LIN {X 0,Y 445.736,Z 432.603,A -85,B 0,C 180,E1 -8644.071,E2 -8644.071} C_VEL
LIN {X 0,Y 445.822,Z 429.975,A -85,B 0,C 180,E1 -8644.977,E2 -8644.977} C_VEL
LIN {X 0,Y 445.879,Z 426.705,A -85,B 0,C 180,E1 -8645.883,E2 -8645.883} C_VEL
LIN {X 0,Y 446.166,Z 422.759,A -85,B 0,C 180,E1 -8646.774,E2 -8646.774} C_VEL
LIN {X 0,Y 446.258,Z 417.856,A -85,B 0,C 180,E1 -8647.696,E2 -8647.696} C_VEL
LIN {X 0,Y 446.578,Z 411.998,A -85,B 0,C 180,E1 -8648.601,E2 -8648.601} C_VEL
LIN {X 0,Y 446.917,Z 404.901,A -85,B 0,C 180,E1 -8649.507,E2 -8649.507} C_VEL
LIN {X 0,Y 447.271,Z 396.212,A -85,B 0,C 180,E1 -8650.413,E2 -8650.413} C_VEL
LIN {X 0,Y 447.669,Z 386.58,A -85,B 0,C 180,E1 -8651.205,E2 -8651.205} C_VEL
LIN {X 0,Y 447.943,Z 376.584,A -85,B 0,C 180,E1 -8651.829,E2 -8651.829} C_VEL
LIN {X 0,Y 448.145,Z 366.978,A -85,B 0,C 180,E1 -8652.283,E2 -8652.283} C_VEL
LIN {X 0,Y 448.381,Z 355.812,A -85,B 0,C 180,E1 -8652.65,E2 -8652.65} C_VEL
LIN {X 0,Y 449.184,Z 291.392,A -85,B 0,C 180,E1 -8653.927,E2 -8653.927} C_VEL
LIN {X 0,Y 446.83,Z 279.728,A -85,B 0,C 180,E1 -8654.297,E2 -8654.297} C_VEL
LIN {X 0,Y 446.931,Z 267.696,A -85,B 0,C 180,E1 -8657.151,E2 -8657.151} C_VEL
LIN {X 0,Y 446.52,Z 264.687,A -85,B 0,C 180,E1 -8657.935,E2 -8657.935} C_VEL
LIN {X 0,Y 446.462,Z 264.684,A -85,B 0,C 180,E1 -8661.229,E2 -8661.229} C_VEL
LIN {X 0,Y 446.469,Z 264.688,A -85,B 0,C 180,E1 -8664.161,E2 -8664.161} C_VEL
LIN {X 0,Y 446.45,Z 264.685,A -85,B 0,C 180,E1 -8667.165,E2 -8667.165} C_VEL
LIN {X 0,Y 446.434,Z 264.691,A -85,B 0,C 180,E1 -8670.251,E2 -8670.251} C_VEL
LIN {X 0,Y 446.433,Z 264.686,A -85,B 0,C 180,E1 -8673.451,E2 -8673.451} C_VEL
LIN {X 0,Y 446.408,Z 264.693,A -85,B 0,C 180,E1 -8676.747,E2 -8676.747} C_VEL
LIN {X 0,Y 446.409,Z 264.688,A -85,B 0,C 180,E1 -8679.517,E2 -8679.517} C_VEL
LIN {X 0,Y 446.424,Z 264.691,A -85,B 0,C 180,E1 -8682.607,E2 -8682.607} C_VEL
LIN {X 0,Y 446.459,Z 264.682,A -85,B 0,C 180,E1 -8685.105,E2 -8685.105} C_VEL
LIN {X 0,Y 446.427,Z 264.69,A -85,B 0,C 180,E1 -8688.608,E2 -8688.608} C_VEL
LIN {X 0,Y 446.418,Z 264.687,A -85,B 0,C 180,E1 -8691.922,E2 -8691.922} C_VEL
LIN {X 0,Y 446.429,Z 264.685,A -85,B 0,C 180,E1 -8695.477,E2 -8695.477} C_VEL
LIN {X 0,Y 446.422,Z 264.689,A -85,B 0,C 180,E1 -8698.7,E2 -8698.7} C_VEL
LIN {X 0,Y 446.493,Z 264.679,A -85,B 0,C 180,E1 -8701.822,E2 -8701.822} C_VEL
LIN {X 0,Y 446.529,Z 264.791,A -85,B 0,C 180,E1 -8705.349,E2 -8705.349} C_VEL
LIN {X 0,Y 447.897,Z 273.343,A -85,B 0,C 180,E1 -8707.172,E2 -8707.172} C_VEL
LIN {X 0,Y 447.39,Z 287.311,A -85,B 0,C 180,E1 -8710.005,E2 -8710.005} C_VEL
LIN {X 0,Y 446.674,Z 303.817,A -85,B 0,C 180,E1 -8713.313,E2 -8713.313} C_VEL
LIN {X 0,Y 446.274,Z 317.421,A -85,B 0,C 180,E1 -8716.017,E2 -8716.017} C_VEL
LIN {X 0,Y 448.11,Z 333.386,A -85,B 0,C 180,E1 -8716.393,E2 -8716.393} C_VEL
LIN {X 0,Y 448.546,Z 340.204,A -85,B 0,C 180,E1 -8716.515,E2 -8716.515} C_VEL
LIN {X 0,Y 448.123,Z 395.887,A -85,B 0,C 180,E1 -8717.431,E2 -8717.431} C_VEL
LIN {X 0,Y 447.824,Z 406.318,A -85,B 0,C 180,E1 -8717.739,E2 -8717.739} C_VEL
LIN {X 0,Y 447.468,Z 417.027,A -85,B 0,C 180,E1 -8718.218,E2 -8718.218} C_VEL
LIN {X 0,Y 447.098,Z 427.678,A -85,B 0,C 180,E1 -8718.898,E2 -8718.898} C_VEL
LIN {X 0,Y 446.741,Z 436.021,A -85,B 0,C 180,E1 -8719.577,E2 -8719.577} C_VEL
LIN {X 0,Y 446.432,Z 443.922,A -85,B 0,C 180,E1 -8720.371,E2 -8720.371} C_VEL
LIN {X 0,Y 446.124,Z 450.448,A -85,B 0,C 180,E1 -8721.164,E2 -8721.164} C_VEL
LIN {X 0,Y 445.865,Z 456.661,A -85,B 0,C 180,E1 -8722.072,E2 -8722.072} C_VEL
LIN {X 0,Y 445.732,Z 461.938,A -85,B 0,C 180,E1 -8723.004,E2 -8723.004} C_VEL
LIN {X 0,Y 445.526,Z 467.071,A -85,B 0,C 180,E1 -8724.115,E2 -8724.115} C_VEL
LIN {X 0,Y 445.436,Z 471.949,A -85,B 0,C 180,E1 -8725.475,E2 -8725.475} C_VEL
LIN {X 0,Y 445.445,Z 474.326,A -85,B 0,C 180,E1 -8726.381,E2 -8726.381} C_VEL
LIN {X 0,Y 445.461,Z 476.147,A -85,B 0,C 180,E1 -8727.287,E2 -8727.287} C_VEL
LIN {X 0,Y 445.401,Z 477.46,A -85,B 0,C 180,E1 -8728.191,E2 -8728.191} C_VEL
LIN {X 0,Y 445.398,Z 478.295,A -85,B 0,C 180,E1 -8729.096,E2 -8729.096} C_VEL
LIN {X 0,Y 445.406,Z 478.604,A -85,B 0,C 180,E1 -8730,E2 -8730} C_VEL
LIN {X 0,Y 445.383,Z 478.332,A -85,B 0,C 180,E1 -8730.904,E2 -8730.904} C_VEL
LIN {X 0,Y 445.401,Z 477.593,A -85,B 0,C 180,E1 -8731.808,E2 -8731.808} C_VEL
LIN {X 0,Y 445.461,Z 476.38,A -85,B 0,C 180,E1 -8732.713,E2 -8732.713} C_VEL
LIN {X 0,Y 445.413,Z 473.501,A -85,B 0,C 180,E1 -8734.071,E2 -8734.071} C_VEL
LIN {X 0,Y 445.536,Z 469.363,A -85,B 0,C 180,E1 -8735.431,E2 -8735.431} C_VEL
LIN {X 0,Y 445.709,Z 463.763,A -85,B 0,C 180,E1 -8736.791,E2 -8736.791} C_VEL
LIN {X 0,Y 445.901,Z 457.634,A -85,B 0,C 180,E1 -8737.927,E2 -8737.927} C_VEL
LIN {X 0,Y 446.159,Z 451.67,A -85,B 0,C 180,E1 -8738.835,E2 -8738.835} C_VEL
LIN {X 0,Y 446.529,Z 444.423,A -85,B 0,C 180,E1 -8739.741,E2 -8739.741} C_VEL
LIN {X 0,Y 446.901,Z 436.704,A -85,B 0,C 180,E1 -8740.534,E2 -8740.534} C_VEL
LIN {X 0,Y 447.199,Z 430.1,A -85,B 0,C 180,E1 -8741.099,E2 -8741.099} C_VEL
LIN {X 0,Y 447.529,Z 422.072,A -85,B 0,C 180,E1 -8741.665,E2 -8741.665} C_VEL
LIN {X 0,Y 447.862,Z 412.829,A -85,B 0,C 180,E1 -8742.173,E2 -8742.173} C_VEL
LIN {X 0,Y 448.205,Z 403.867,A -85,B 0,C 180,E1 -8742.537,E2 -8742.537} C_VEL
LIN {X 0,Y 448.527,Z 394.863,A -85,B 0,C 180,E1 -8742.786,E2 -8742.786} C_VEL
LIN {X 0,Y 448.842,Z 336.982,A -85,B 0,C 180,E1 -8743.748,E2 -8743.748} C_VEL
LIN {X 0,Y 446.374,Z 317.409,A -85,B 0,C 180,E1 -8744.161,E2 -8744.161} C_VEL
LIN {X 0,Y 446.932,Z 300.088,A -85,B 0,C 180,E1 -8747.62,E2 -8747.62} C_VEL
LIN {X 0,Y 447.632,Z 284.911,A -85,B 0,C 180,E1 -8750.687,E2 -8750.687} C_VEL
LIN {X 0,Y 448.083,Z 274.39,A -85,B 0,C 180,E1 -8752.842,E2 -8752.842} C_VEL
LIN {X 0,Y 446.746,Z 266.156,A -85,B 0,C 180,E1 -8754.637,E2 -8754.637} C_VEL
LIN {X 0,Y 446.479,Z 264.685,A -85,B 0,C 180,E1 -8754.995,E2 -8754.995} C_VEL
LIN {X 0,Y 446.492,Z 264.679,A -85,B 0,C 180,E1 -8758.178,E2 -8758.178} C_VEL
LIN {X 0,Y 446.422,Z 264.685,A -85,B 0,C 180,E1 -8761.773,E2 -8761.773} C_VEL
LIN {X 0,Y 446.428,Z 264.687,A -85,B 0,C 180,E1 -8764.523,E2 -8764.523} C_VEL
LIN {X 0,Y 446.419,Z 264.687,A -85,B 0,C 180,E1 -8768.078,E2 -8768.078} C_VEL
LIN {X 0,Y 446.426,Z 264.69,A -85,B 0,C 180,E1 -8771.391,E2 -8771.391} C_VEL
LIN {X 0,Y 446.457,Z 264.682,A -85,B 0,C 180,E1 -8775.103,E2 -8775.103} C_VEL
LIN {X 0,Y 446.425,Z 264.685,A -85,B 0,C 180,E1 -8778.607,E2 -8778.607} C_VEL
LIN {X 0,Y 446.418,Z 264.689,A -85,B 0,C 180,E1 -8781.92,E2 -8781.92} C_VEL
LIN {X 0,Y 446.43,Z 264.686,A -85,B 0,C 180,E1 -8785.475,E2 -8785.475} C_VEL
LIN {X 0,Y 446.421,Z 264.682,A -85,B 0,C 180,E1 -8788.698,E2 -8788.698} C_VEL
LIN {X 0,Y 446.455,Z 264.686,A -85,B 0,C 180,E1 -8791.828,E2 -8791.828} C_VEL
LIN {X 0,Y 446.449,Z 264.68,A -85,B 0,C 180,E1 -8794.845,E2 -8794.845} C_VEL
LIN {X 0,Y 446.454,Z 264.678,A -85,B 0,C 180,E1 -8798.243,E2 -8798.243} C_VEL
LIN {X 0,Y 446.457,Z 264.686,A -85,B 0,C 180,E1 -8801.647,E2 -8801.647} C_VEL
LIN {X 0,Y 446.512,Z 264.672,A -85,B 0,C 180,E1 -8804.478,E2 -8804.478} C_VEL
LIN {X 0,Y 446.521,Z 264.67,A -85,B 0,C 180,E1 -8808.191,E2 -8808.191} C_VEL
LIN {X 0,Y 446.603,Z 264.666,A -85,B 0,C 180,E1 -8811.855,E2 -8811.855} C_VEL
LIN {X 0,Y 446.644,Z 264.652,A -85,B 0,C 180,E1 -8814.58,E2 -8814.58} C_VEL
LIN {X 0,Y 446.662,Z 264.656,A -85,B 0,C 180,E1 -8818.194,E2 -8818.194} C_VEL
LIN {X 0,Y 446.789,Z 264.638,A -85,B 0,C 180,E1 -8819.997,E2 -8819.997} C_VEL
LIN {X 0,Y 446.682,Z 264.652,A -85,B 0,C 180,E1 -8822.702,E2 -8822.702} C_VEL
LIN {X 0,Y 446.614,Z 264.664,A -85,B 0,C 180,E1 -8826.321,E2 -8826.321} C_VEL
LIN {X 0,Y 446.529,Z 264.67,A -85,B 0,C 180,E1 -8829.052,E2 -8829.052} C_VEL
LIN {X 0,Y 446.516,Z 264.676,A -85,B 0,C 180,E1 -8832.726,E2 -8832.726} C_VEL
LIN {X 0,Y 446.488,Z 264.678,A -85,B 0,C 180,E1 -8836.224,E2 -8836.224} C_VEL
LIN {X 0,Y 446.459,Z 264.679,A -85,B 0,C 180,E1 -8839.3,E2 -8839.3} C_VEL
LIN {X 0,Y 446.408,Z 264.691,A -85,B 0,C 180,E1 -8842.196,E2 -8842.196} C_VEL
LIN {X 0,Y 446.445,Z 264.682,A -85,B 0,C 180,E1 -8845.149,E2 -8845.149} C_VEL
LIN {X 0,Y 446.47,Z 264.683,A -85,B 0,C 180,E1 -8848.175,E2 -8848.175} C_VEL
LIN {X 0,Y 446.402,Z 264.686,A -85,B 0,C 180,E1 -8851.772,E2 -8851.772} C_VEL
LIN {X 0,Y 446.412,Z 264.689,A -85,B 0,C 180,E1 -8854.52,E2 -8854.52} C_VEL
LIN {X 0,Y 446.395,Z 264.691,A -85,B 0,C 180,E1 -8858.076,E2 -8858.076} C_VEL
LIN {X 0,Y 446.409,Z 264.69,A -85,B 0,C 180,E1 -8860.915,E2 -8860.915} C_VEL
LIN {X 0,Y 446.422,Z 264.685,A -85,B 0,C 180,E1 -8863.837,E2 -8863.837} C_VEL
LIN {X 0,Y 446.422,Z 264.691,A -85,B 0,C 180,E1 -8866.394,E2 -8866.394} C_VEL
LIN {X 0,Y 446.442,Z 264.685,A -85,B 0,C 180,E1 -8869.802,E2 -8869.802} C_VEL
LIN {X 0,Y 446.407,Z 264.692,A -85,B 0,C 180,E1 -8872.121,E2 -8872.121} C_VEL
LIN {X 0,Y 446.467,Z 264.833,A -85,B 0,C 180,E1 -8875.58,E2 -8875.58} C_VEL
LIN {X 0,Y 446.785,Z 269.023,A -85,B 0,C 180,E1 -8876.595,E2 -8876.595} C_VEL
LIN {X 0,Y 446.663,Z 278.985,A -85,B 0,C 180,E1 -8878.905,E2 -8878.905} C_VEL
LIN {X 0,Y 449.203,Z 291.834,A -85,B 0,C 180,E1 -8879.21,E2 -8879.21} C_VEL
LIN {X 0,Y 448.652,Z 354.384,A -85,B 0,C 180,E1 -8880.24,E2 -8880.24} C_VEL
LIN {X 0,Y 448.492,Z 364.23,A -85,B 0,C 180,E1 -8880.518,E2 -8880.518} C_VEL
LIN {X 0,Y 448.303,Z 373.791,A -85,B 0,C 180,E1 -8880.923,E2 -8880.923} C_VEL
LIN {X 0,Y 447.973,Z 384.881,A -85,B 0,C 180,E1 -8881.57,E2 -8881.57} C_VEL
LIN {X 0,Y 447.591,Z 393.904,A -85,B 0,C 180,E1 -8882.279,E2 -8882.279} C_VEL
LIN {X 0,Y 447.127,Z 402.361,A -85,B 0,C 180,E1 -8883.112,E2 -8883.112} C_VEL
LIN {X 0,Y 446.836,Z 408.702,A -85,B 0,C 180,E1 -8883.871,E2 -8883.871} C_VEL
LIN {X 0,Y 446.472,Z 415.446,A -85,B 0,C 180,E1 -8884.849,E2 -8884.849} C_VEL
LIN {X 0,Y 446.21,Z 420.965,A -85,B 0,C 180,E1 -8885.826,E2 -8885.826} C_VEL
LIN {X 0,Y 445.956,Z 425.477,A -85,B 0,C 180,E1 -8886.797,E2 -8886.797} C_VEL
LIN {X 0,Y 445.751,Z 429.838,A -85,B 0,C 180,E1 -8887.976,E2 -8887.976} C_VEL
LIN {X 0,Y 445.602,Z 433.289,A -85,B 0,C 180,E1 -8889.215,E2 -8889.215} C_VEL
LIN {X 0,Y 445.44,Z 436.017,A -85,B 0,C 180,E1 -8890.651,E2 -8890.651} C_VEL
LIN {X 0,Y 445.362,Z 437.127,A -85,B 0,C 180,E1 -8891.788,E2 -8891.788} C_VEL
LIN {X 0,Y 444.655,Z 437.549,A -85,B 0,C 180,E1 -8892.543,E2 -8892.543} C_VEL
LIN {X 0,Y 441.789,Z 437.502,A -85,B 0,C 180,E1 -8893.771,E2 -8893.771} C_VEL
LIN {X 0,Y 439.413,Z 436.81,A -85,B 0,C 180,E1 -8894.756,E2 -8894.756} C_VEL
LIN {X 0,Y 438.424,Z 435.902,A -85,B 0,C 180,E1 -8895.51,E2 -8895.51} C_VEL
LIN {X 0,Y 438.359,Z 435.425,A -85,B 0,C 180,E1 -8895.763,E2 -8895.763} C_VEL
LIN {X 0,Y 438.477,Z 432.779,A -85,B 0,C 180,E1 -8897.033,E2 -8897.033} C_VEL
LIN {X 0,Y 438.625,Z 430.078,A -85,B 0,C 180,E1 -8897.978,E2 -8897.978} C_VEL
LIN {X 0,Y 438.845,Z 424.796,A -85,B 0,C 180,E1 -8899.387,E2 -8899.387} C_VEL
LIN {X 0,Y 439.138,Z 417.792,A -85,B 0,C 180,E1 -8900.791,E2 -8900.791} C_VEL
LIN {X 0,Y 439.527,Z 410.412,A -85,B 0,C 180,E1 -8901.92,E2 -8901.92} C_VEL
LIN {X 0,Y 439.807,Z 403.614,A -85,B 0,C 180,E1 -8902.771,E2 -8902.771} C_VEL
LIN {X 0,Y 440.125,Z 396.941,A -85,B 0,C 180,E1 -8903.467,E2 -8903.467} C_VEL
LIN {X 0,Y 440.468,Z 388.851,A -85,B 0,C 180,E1 -8904.162,E2 -8904.162} C_VEL
LIN {X 0,Y 440.768,Z 380.467,A -85,B 0,C 180,E1 -8904.74,E2 -8904.74} C_VEL
LIN {X 0,Y 440.955,Z 371.957,A -85,B 0,C 180,E1 -8905.2,E2 -8905.2} C_VEL
LIN {X 0,Y 441.152,Z 362.617,A -85,B 0,C 180,E1 -8905.574,E2 -8905.574} C_VEL
LIN {X 0,Y 441.314,Z 351.534,A -85,B 0,C 180,E1 -8905.862,E2 -8905.862} C_VEL
LIN {X 0,Y 441.724,Z 291.914,A -85,B 0,C 180,E1 -8906.836,E2 -8906.836} C_VEL
LIN {X 0,Y 439.372,Z 278.971,A -85,B 0,C 180,E1 -8907.135,E2 -8907.135} C_VEL
LIN {X 0,Y 439.691,Z 267.341,A -85,B 0,C 180,E1 -8910,E2 -8910} C_VEL
LIN {X 0,Y 439.584,Z 265.543,A -85,B 0,C 180,E1 -8910.458,E2 -8910.458} C_VEL
LIN {X 0,Y 439.619,Z 265.535,A -85,B 0,C 180,E1 -8912.749,E2 -8912.749} C_VEL
LIN {X 0,Y 439.577,Z 265.538,A -85,B 0,C 180,E1 -8916.426,E2 -8916.426} C_VEL
LIN {X 0,Y 439.463,Z 265.559,A -85,B 0,C 180,E1 -8919.203,E2 -8919.203} C_VEL
LIN {X 0,Y 439.429,Z 265.559,A -85,B 0,C 180,E1 -8922.939,E2 -8922.939} C_VEL
LIN {X 0,Y 439.411,Z 265.558,A -85,B 0,C 180,E1 -8926.35,E2 -8926.35} C_VEL
LIN {X 0,Y 439.367,Z 265.568,A -85,B 0,C 180,E1 -8929.628,E2 -8929.628} C_VEL
LIN {X 0,Y 439.328,Z 265.568,A -85,B 0,C 180,E1 -8932.578,E2 -8932.578} C_VEL
LIN {X 0,Y 439.344,Z 265.572,A -85,B 0,C 180,E1 -8935.589,E2 -8935.589} C_VEL
LIN {X 0,Y 439.365,Z 265.564,A -85,B 0,C 180,E1 -8938.677,E2 -8938.677} C_VEL
LIN {X 0,Y 439.339,Z 265.569,A -85,B 0,C 180,E1 -8942.033,E2 -8942.033} C_VEL
LIN {X 0,Y 439.364,Z 265.569,A -85,B 0,C 180,E1 -8945.343,E2 -8945.343} C_VEL
LIN {X 0,Y 439.334,Z 265.568,A -85,B 0,C 180,E1 -8948.6,E2 -8948.6} C_VEL
LIN {X 0,Y 439.357,Z 265.566,A -85,B 0,C 180,E1 -8952.209,E2 -8952.209} C_VEL
LIN {X 0,Y 439.376,Z 265.566,A -85,B 0,C 180,E1 -8955.274,E2 -8955.274} C_VEL
LIN {X 0,Y 439.368,Z 265.564,A -85,B 0,C 180,E1 -8958.747,E2 -8958.747} C_VEL
LIN {X 0,Y 439.35,Z 265.572,A -85,B 0,C 180,E1 -8961.612,E2 -8961.612} C_VEL
LIN {X 0,Y 439.379,Z 265.563,A -85,B 0,C 180,E1 -8964.847,E2 -8964.847} C_VEL
LIN {X 0,Y 439.357,Z 265.569,A -85,B 0,C 180,E1 -8968.143,E2 -8968.143} C_VEL
LIN {X 0,Y 439.396,Z 265.565,A -85,B 0,C 180,E1 -8971.608,E2 -8971.608} C_VEL
LIN {X 0,Y 439.365,Z 265.566,A -85,B 0,C 180,E1 -8974.417,E2 -8974.417} C_VEL
LIN {X 0,Y 439.355,Z 265.568,A -85,B 0,C 180,E1 -8977.428,E2 -8977.428} C_VEL
LIN {X 0,Y 439.434,Z 265.557,A -85,B 0,C 180,E1 -8980.667,E2 -8980.667} C_VEL
LIN {X 0,Y 439.488,Z 265.678,A -85,B 0,C 180,E1 -8982.916,E2 -8982.916} C_VEL
LIN {X 0,Y 439.373,Z 276.791,A -85,B 0,C 180,E1 -8985.648,E2 -8985.648} C_VEL
LIN {X 0,Y 439.369,Z 278.594,A -85,B 0,C 180,E1 -8986.091,E2 -8986.091} C_VEL
LIN {X 0,Y 441.507,Z 292.814,A -85,B 0,C 180,E1 -8986.425,E2 -8986.425} C_VEL
LIN {X 0,Y 440.848,Z 355.577,A -85,B 0,C 180,E1 -8987.634,E2 -8987.634} C_VEL
LIN {X 0,Y 440.64,Z 366.074,A -85,B 0,C 180,E1 -8987.978,E2 -8987.978} C_VEL
LIN {X 0,Y 440.366,Z 375.868,A -85,B 0,C 180,E1 -8988.438,E2 -8988.438} C_VEL
LIN {X 0,Y 440.199,Z 386.05,A -85,B 0,C 180,E1 -8989.075,E2 -8989.075} C_VEL
LIN {X 0,Y 439.835,Z 395.801,A -85,B 0,C 180,E1 -8989.88,E2 -8989.88} C_VEL
LIN {X 0,Y 439.545,Z 403.626,A -85,B 0,C 180,E1 -8990.687,E2 -8990.687} C_VEL
LIN {X 0,Y 439.192,Z 411.811,A -85,B 0,C 180,E1 -8991.723,E2 -8991.723} C_VEL
LIN {X 0,Y 439.012,Z 419.739,A -85,B 0,C 180,E1 -8992.998,E2 -8992.998} C_VEL
LIN {X 0,Y 438.774,Z 424.777,A -85,B 0,C 180,E1 -8994.027,E2 -8994.027} C_VEL
LIN {X 0,Y 438.578,Z 430.038,A -85,B 0,C 180,E1 -8995.408,E2 -8995.408} C_VEL
LIN {X 0,Y 438.563,Z 432.715,A -85,B 0,C 180,E1 -8996.328,E2 -8996.328} C_VEL
LIN {X 0,Y 438.454,Z 434.806,A -85,B 0,C 180,E1 -8997.247,E2 -8997.247} C_VEL
LIN {X 0,Y 438.353,Z 436.351,A -85,B 0,C 180,E1 -8998.165,E2 -8998.165} C_VEL
LIN {X 0,Y 438.313,Z 437.348,A -85,B 0,C 180,E1 -8999.084,E2 -8999.084} C_VEL
LIN {X 0,Y 438.318,Z 437.751,A -85,B 0,C 180,E1 -9000.003,E2 -9000.003} C_VEL
LIN {X 0,Y 438.344,Z 437.622,A -85,B 0,C 180,E1 -9000.922,E2 -9000.922} C_VEL
LIN {X 0,Y 438.393,Z 436.987,A -85,B 0,C 180,E1 -9001.84,E2 -9001.84} C_VEL
LIN {X 0,Y 438.483,Z 435.838,A -85,B 0,C 180,E1 -9002.759,E2 -9002.759} C_VEL
LIN {X 0,Y 438.686,Z 433.017,A -85,B 0,C 180,E1 -9004.137,E2 -9004.137} C_VEL
LIN {X 0,Y 438.768,Z 430.415,A -85,B 0,C 180,E1 -9005.057,E2 -9005.057} C_VEL
LIN {X 0,Y 438.848,Z 427.178,A -85,B 0,C 180,E1 -9005.978,E2 -9005.978} C_VEL
LIN {X 0,Y 439.143,Z 422.003,A -85,B 0,C 180,E1 -9007.14,E2 -9007.14} C_VEL
LIN {X 0,Y 439.334,Z 417.041,A -85,B 0,C 180,E1 -9008.049,E2 -9008.049} C_VEL
LIN {X 0,Y 439.645,Z 410.982,A -85,B 0,C 180,E1 -9008.969,E2 -9008.969} C_VEL
LIN {X 0,Y 440.092,Z 402.644,A -85,B 0,C 180,E1 -9010.004,E2 -9010.004} C_VEL
LIN {X 0,Y 440.515,Z 393.123,A -85,B 0,C 180,E1 -9010.924,E2 -9010.924} C_VEL
LIN {X 0,Y 440.857,Z 384.062,A -85,B 0,C 180,E1 -9011.613,E2 -9011.613} C_VEL
LIN {X 0,Y 441.16,Z 373.345,A -85,B 0,C 180,E1 -9012.247,E2 -9012.247} C_VEL
LIN {X 0,Y 441.416,Z 361.296,A -85,B 0,C 180,E1 -9012.736,E2 -9012.736} C_VEL
LIN {X 0,Y 441.682,Z 350.319,A -85,B 0,C 180,E1 -9013.013,E2 -9013.013} C_VEL
LIN {X 0,Y 442.48,Z 292.448,A -85,B 0,C 180,E1 -9014.193,E2 -9014.193} C_VEL
LIN {X 0,Y 439.876,Z 280.051,A -85,B 0,C 180,E1 -9014.601,E2 -9014.601} C_VEL
LIN {X 0,Y 440.016,Z 269.226,A -85,B 0,C 180,E1 -9017.189,E2 -9017.189} C_VEL
LIN {X 0,Y 439.487,Z 265.563,A -85,B 0,C 180,E1 -9018.112,E2 -9018.112} C_VEL
LIN {X 0,Y 439.424,Z 265.561,A -85,B 0,C 180,E1 -9021.586,E2 -9021.586} C_VEL
LIN {X 0,Y 439.414,Z 265.564,A -85,B 0,C 180,E1 -9024.575,E2 -9024.575} C_VEL
LIN {X 0,Y 439.392,Z 265.565,A -85,B 0,C 180,E1 -9027.638,E2 -9027.638} C_VEL
LIN {X 0,Y 439.369,Z 265.569,A -85,B 0,C 180,E1 -9030.79,E2 -9030.79} C_VEL
LIN {X 0,Y 439.368,Z 265.569,A -85,B 0,C 180,E1 -9034.048,E2 -9034.048} C_VEL
LIN {X 0,Y 439.355,Z 265.57,A -85,B 0,C 180,E1 -9036.888,E2 -9036.888} C_VEL
LIN {X 0,Y 439.356,Z 265.568,A -85,B 0,C 180,E1 -9039.842,E2 -9039.842} C_VEL
LIN {X 0,Y 439.378,Z 265.568,A -85,B 0,C 180,E1 -9042.626,E2 -9042.626} C_VEL
LIN {X 0,Y 439.407,Z 265.56,A -85,B 0,C 180,E1 -9045.271,E2 -9045.271} C_VEL
LIN {X 0,Y 439.39,Z 265.566,A -85,B 0,C 180,E1 -9048.745,E2 -9048.745} C_VEL
LIN {X 0,Y 439.373,Z 265.564,A -85,B 0,C 180,E1 -9051.61,E2 -9051.61} C_VEL
LIN {X 0,Y 439.403,Z 265.565,A -85,B 0,C 180,E1 -9054.844,E2 -9054.844} C_VEL
LIN {X 0,Y 439.377,Z 265.566,A -85,B 0,C 180,E1 -9058.14,E2 -9058.14} C_VEL
LIN {X 0,Y 439.441,Z 265.557,A -85,B 0,C 180,E1 -9061.599,E2 -9061.599} C_VEL
LIN {X 0,Y 439.476,Z 265.609,A -85,B 0,C 180,E1 -9065.21,E2 -9065.21} C_VEL
LIN {X 0,Y 440.873,Z 273.902,A -85,B 0,C 180,E1 -9067.011,E2 -9067.011} C_VEL
LIN {X 0,Y 440.524,Z 283.37,A -85,B 0,C 180,E1 -9068.963,E2 -9068.963} C_VEL
LIN {X 0,Y 439.86,Z 298.668,A -85,B 0,C 180,E1 -9072.087,E2 -9072.087} C_VEL
LIN {X 0,Y 439.252,Z 316.225,A -85,B 0,C 180,E1 -9075.641,E2 -9075.641} C_VEL
LIN {X 0,Y 439.233,Z 316.568,A -85,B 0,C 180,E1 -9075.699,E2 -9075.699} C_VEL
LIN {X 0,Y 441.57,Z 337.97,A -85,B 0,C 180,E1 -9076.27,E2 -9076.27} C_VEL
LIN {X 0,Y 441.16,Z 395.561,A -85,B 0,C 180,E1 -9077.259,E2 -9077.259} C_VEL
LIN {X 0,Y 440.856,Z 405.999,A -85,B 0,C 180,E1 -9077.572,E2 -9077.572} C_VEL
LIN {X 0,Y 440.431,Z 418.159,A -85,B 0,C 180,E1 -9078.144,E2 -9078.144} C_VEL
LIN {X 0,Y 440.087,Z 426.992,A -85,B 0,C 180,E1 -9078.718,E2 -9078.718} C_VEL
LIN {X 0,Y 439.737,Z 435.409,A -85,B 0,C 180,E1 -9079.409,E2 -9079.409} C_VEL
LIN {X 0,Y 439.399,Z 443.365,A -85,B 0,C 180,E1 -9080.215,E2 -9080.215} C_VEL
LIN {X 0,Y 439.098,Z 449.935,A -85,B 0,C 180,E1 -9081.022,E2 -9081.022} C_VEL
LIN {X 0,Y 438.794,Z 456.182,A -85,B 0,C 180,E1 -9081.944,E2 -9081.944} C_VEL
LIN {X 0,Y 438.673,Z 461.373,A -85,B 0,C 180,E1 -9082.867,E2 -9082.867} C_VEL
LIN {X 0,Y 438.449,Z 466.163,A -85,B 0,C 180,E1 -9083.903,E2 -9083.903} C_VEL
LIN {X 0,Y 438.443,Z 470.034,A -85,B 0,C 180,E1 -9084.942,E2 -9084.942} C_VEL
LIN {X 0,Y 438.326,Z 472.781,A -85,B 0,C 180,E1 -9085.862,E2 -9085.862} C_VEL
LIN {X 0,Y 438.388,Z 475.783,A -85,B 0,C 180,E1 -9087.243,E2 -9087.243} C_VEL
LIN {X 0,Y 438.321,Z 477.111,A -85,B 0,C 180,E1 -9088.162,E2 -9088.162} C_VEL
LIN {X 0,Y 438.308,Z 477.961,A -85,B 0,C 180,E1 -9089.081,E2 -9089.081} C_VEL
LIN {X 0,Y 438.314,Z 478.272,A -85,B 0,C 180,E1 -9090,E2 -9090} C_VEL
LIN {X 0,Y 438.294,Z 478.012,A -85,B 0,C 180,E1 -9090.919,E2 -9090.919} C_VEL
LIN {X 0,Y 438.321,Z 477.287,A -85,B 0,C 180,E1 -9091.837,E2 -9091.837} C_VEL
LIN {X 0,Y 438.387,Z 476.09,A -85,B 0,C 180,E1 -9092.756,E2 -9092.756} C_VEL
LIN {X 0,Y 438.325,Z 473.228,A -85,B 0,C 180,E1 -9094.137,E2 -9094.137} C_VEL
LIN {X 0,Y 438.432,Z 469.11,A -85,B 0,C 180,E1 -9095.519,E2 -9095.519} C_VEL
LIN {X 0,Y 438.666,Z 463.551,A -85,B 0,C 180,E1 -9096.901,E2 -9096.901} C_VEL
LIN {X 0,Y 438.849,Z 457.466,A -85,B 0,C 180,E1 -9098.055,E2 -9098.055} C_VEL
LIN {X 0,Y 439.13,Z 451.543,A -85,B 0,C 180,E1 -9098.977,E2 -9098.977} C_VEL
LIN {X 0,Y 439.525,Z 444.346,A -85,B 0,C 180,E1 -9099.898,E2 -9099.898} C_VEL
LIN {X 0,Y 439.925,Z 436.678,A -85,B 0,C 180,E1 -9100.703,E2 -9100.703} C_VEL
LIN {X 0,Y 440.316,Z 428.641,A -85,B 0,C 180,E1 -9101.392,E2 -9101.392} C_VEL
LIN {X 0,Y 440.651,Z 420.335,A -85,B 0,C 180,E1 -9101.966,E2 -9101.966} C_VEL
LIN {X 0,Y 441.007,Z 411.891,A -85,B 0,C 180,E1 -9102.424,E2 -9102.424} C_VEL
LIN {X 0,Y 441.359,Z 402.705,A -85,B 0,C 180,E1 -9102.793,E2 -9102.793} C_VEL
LIN {X 0,Y 441.629,Z 392.454,A -85,B 0,C 180,E1 -9103.066,E2 -9103.066} C_VEL
LIN {X 0,Y 441.941,Z 337.18,A -85,B 0,C 180,E1 -9103.988,E2 -9103.988} C_VEL
LIN {X 0,Y 439.62,Z 318.849,A -85,B 0,C 180,E1 -9104.38,E2 -9104.38} C_VEL
LIN {X 0,Y 439.355,Z 316.991,A -85,B 0,C 180,E1 -9104.438,E2 -9104.438} C_VEL
LIN {X 0,Y 439.917,Z 301.084,A -85,B 0,C 180,E1 -9107.67,E2 -9107.67} C_VEL
LIN {X 0,Y 440.652,Z 285.919,A -85,B 0,C 180,E1 -9110.785,E2 -9110.785} C_VEL
LIN {X 0,Y 441.11,Z 275.395,A -85,B 0,C 180,E1 -9112.976,E2 -9112.976} C_VEL
LIN {X 0,Y 439.426,Z 265.564,A -85,B 0,C 180,E1 -9115.203,E2 -9115.203} C_VEL
LIN {X 0,Y 439.439,Z 265.558,A -85,B 0,C 180,E1 -9118.401,E2 -9118.401} C_VEL
LIN {X 0,Y 439.375,Z 265.562,A -85,B 0,C 180,E1 -9121.86,E2 -9121.86} C_VEL
LIN {X 0,Y 439.398,Z 265.561,A -85,B 0,C 180,E1 -9125.339,E2 -9125.339} C_VEL
LIN {X 0,Y 439.37,Z 265.565,A -85,B 0,C 180,E1 -9128.596,E2 -9128.596} C_VEL
LIN {X 0,Y 439.389,Z 265.566,A -85,B 0,C 180,E1 -9131.255,E2 -9131.255} C_VEL
LIN {X 0,Y 439.405,Z 265.558,A -85,B 0,C 180,E1 -9134.729,E2 -9134.729} C_VEL
LIN {X 0,Y 439.391,Z 265.565,A -85,B 0,C 180,E1 -9137.793,E2 -9137.793} C_VEL
LIN {X 0,Y 439.365,Z 265.563,A -85,B 0,C 180,E1 -9140.219,E2 -9140.219} C_VEL
LIN {X 0,Y 439.38,Z 265.565,A -85,B 0,C 180,E1 -9143.711,E2 -9143.711} C_VEL
LIN {X 0,Y 439.378,Z 265.564,A -85,B 0,C 180,E1 -9147.052,E2 -9147.052} C_VEL
LIN {X 0,Y 439.383,Z 265.563,A -85,B 0,C 180,E1 -9150.272,E2 -9150.272} C_VEL
LIN {X 0,Y 439.389,Z 265.563,A -85,B 0,C 180,E1 -9153.391,E2 -9153.391} C_VEL
LIN {X 0,Y 439.389,Z 265.562,A -85,B 0,C 180,E1 -9156.427,E2 -9156.427} C_VEL
LIN {X 0,Y 439.393,Z 265.558,A -85,B 0,C 180,E1 -9159.395,E2 -9159.395} C_VEL
LIN {X 0,Y 439.41,Z 265.558,A -85,B 0,C 180,E1 -9162.306,E2 -9162.306} C_VEL
LIN {X 0,Y 439.452,Z 265.55,A -85,B 0,C 180,E1 -9165.172,E2 -9165.172} C_VEL
LIN {X 0,Y 439.487,Z 265.548,A -85,B 0,C 180,E1 -9167.999,E2 -9167.999} C_VEL
LIN {X 0,Y 439.551,Z 265.543,A -85,B 0,C 180,E1 -9171.724,E2 -9171.724} C_VEL
LIN {X 0,Y 439.62,Z 265.528,A -85,B 0,C 180,E1 -9174.493,E2 -9174.493} C_VEL
LIN {X 0,Y 439.632,Z 265.532,A -85,B 0,C 180,E1 -9178.165,E2 -9178.165} C_VEL
LIN {X 0,Y 439.759,Z 265.513,A -85,B 0,C 180,E1 -9179.997,E2 -9179.997} C_VEL
LIN {X 0,Y 439.632,Z 265.53,A -85,B 0,C 180,E1 -9182.746,E2 -9182.746} C_VEL
LIN {X 0,Y 439.586,Z 265.54,A -85,B 0,C 180,E1 -9186.422,E2 -9186.422} C_VEL
LIN {X 0,Y 439.492,Z 265.546,A -85,B 0,C 180,E1 -9189.198,E2 -9189.198} C_VEL
LIN {X 0,Y 439.46,Z 265.553,A -85,B 0,C 180,E1 -9192.934,E2 -9192.934} C_VEL
LIN {X 0,Y 439.439,Z 265.557,A -85,B 0,C 180,E1 -9196.345,E2 -9196.345} C_VEL
LIN {X 0,Y 439.393,Z 265.56,A -85,B 0,C 180,E1 -9199.623,E2 -9199.623} C_VEL
LIN {X 0,Y 439.354,Z 265.571,A -85,B 0,C 180,E1 -9202.572,E2 -9202.572} C_VEL
LIN {X 0,Y 439.392,Z 265.56,A -85,B 0,C 180,E1 -9205.581,E2 -9205.581} C_VEL
LIN {X 0,Y 439.403,Z 265.564,A -85,B 0,C 180,E1 -9208.67,E2 -9208.67} C_VEL
LIN {X 0,Y 439.353,Z 265.566,A -85,B 0,C 180,E1 -9212.027,E2 -9212.027} C_VEL
LIN {X 0,Y 439.377,Z 265.556,A -85,B 0,C 180,E1 -9215.337,E2 -9215.337} C_VEL
LIN {X 0,Y 439.358,Z 265.573,A -85,B 0,C 180,E1 -9218.592,E2 -9218.592} C_VEL
LIN {X 0,Y 439.373,Z 265.566,A -85,B 0,C 180,E1 -9221.255,E2 -9221.255} C_VEL
LIN {X 0,Y 439.386,Z 265.566,A -85,B 0,C 180,E1 -9224.725,E2 -9224.725} C_VEL
LIN {X 0,Y 439.387,Z 265.563,A -85,B 0,C 180,E1 -9227.795,E2 -9227.795} C_VEL
LIN {X 0,Y 439.425,Z 265.561,A -85,B 0,C 180,E1 -9230.227,E2 -9230.227} C_VEL
LIN {X 0,Y 439.349,Z 265.571,A -85,B 0,C 180,E1 -9233.711,E2 -9233.711} C_VEL
LIN {X 0,Y 439.398,Z 265.704,A -85,B 0,C 180,E1 -9235.403,E2 -9235.403} C_VEL
LIN {X 0,Y 439.834,Z 268.832,A -85,B 0,C 180,E1 -9236.182,E2 -9236.182} C_VEL
LIN {X 0,Y 439.667,Z 279.041,A -85,B 0,C 180,E1 -9238.627,E2 -9238.627} C_VEL
LIN {X 0,Y 442.397,Z 292.797,A -85,B 0,C 180,E1 -9238.974,E2 -9238.974} C_VEL
LIN {X 0,Y 441.784,Z 355.466,A -85,B 0,C 180,E1 -9240.025,E2 -9240.025} C_VEL
LIN {X 0,Y 441.615,Z 365.042,A -85,B 0,C 180,E1 -9240.308,E2 -9240.308} C_VEL
LIN {X 0,Y 441.393,Z 375.349,A -85,B 0,C 180,E1 -9240.761,E2 -9240.761} C_VEL
LIN {X 0,Y 441.006,Z 386.29,A -85,B 0,C 180,E1 -9241.44,E2 -9241.44} C_VEL
LIN {X 0,Y 440.632,Z 395.413,A -85,B 0,C 180,E1 -9242.191,E2 -9242.191} C_VEL
LIN {X 0,Y 440.187,Z 402.763,A -85,B 0,C 180,E1 -9242.933,E2 -9242.933} C_VEL
LIN {X 0,Y 439.865,Z 408.923,A -85,B 0,C 180,E1 -9243.68,E2 -9243.68} C_VEL
LIN {X 0,Y 439.493,Z 415.689,A -85,B 0,C 180,E1 -9244.674,E2 -9244.674} C_VEL
LIN {X 0,Y 439.276,Z 419.974,A -85,B 0,C 180,E1 -9245.419,E2 -9245.419} C_VEL
LIN {X 0,Y 438.996,Z 424.735,A -85,B 0,C 180,E1 -9246.408,E2 -9246.408} C_VEL
LIN {X 0,Y 438.777,Z 428.629,A -85,B 0,C 180,E1 -9247.393,E2 -9247.393} C_VEL
LIN {X 0,Y 438.634,Z 431.765,A -85,B 0,C 180,E1 -9248.376,E2 -9248.376} C_VEL
LIN {X 0,Y 438.498,Z 434.18,A -85,B 0,C 180,E1 -9249.354,E2 -9249.354} C_VEL
LIN {X 0,Y 438.378,Z 435.927,A -85,B 0,C 180,E1 -9250.326,E2 -9250.326} C_VEL
LIN {X 0,Y 438.278,Z 437.418,A -85,B 0,C 180,E1 -9251.775,E2 -9251.775} C_VEL
LIN {X 0,Y 438.259,Z 437.858,A -85,B 0,C 180,E1 -9253.223,E2 -9253.223} C_VEL
LIN {X 0,Y 438.327,Z 437.456,A -85,B 0,C 180,E1 -9254.183,E2 -9254.183} C_VEL
LIN {X 0,Y 438.344,Z 436.46,A -85,B 0,C 180,E1 -9255.136,E2 -9255.136} C_VEL
LIN {X 0,Y 438.359,Z 435.425,A -85,B 0,C 180,E1 -9255.763,E2 -9255.763} C_VEL
LIN {X 0,Y 437.75,Z 434.121,A -85,B 0,C 180,E1 -9256.509,E2 -9256.509} C_VEL
LIN {X 0,Y 435.011,Z 431.229,A -85,B 0,C 180,E1 -9257.701,E2 -9257.701} C_VEL
LIN {X 0,Y 432.323,Z 427.492,A -85,B 0,C 180,E1 -9258.867,E2 -9258.867} C_VEL
LIN {X 0,Y 431.816,Z 424.689,A -85,B 0,C 180,E1 -9259.566,E2 -9259.566} C_VEL
LIN {X 0,Y 432.088,Z 418.189,A -85,B 0,C 180,E1 -9260.875,E2 -9260.875} C_VEL
LIN {X 0,Y 432.491,Z 410.694,A -85,B 0,C 180,E1 -9262.04,E2 -9262.04} C_VEL
LIN {X 0,Y 432.776,Z 404.044,A -85,B 0,C 180,E1 -9262.887,E2 -9262.887} C_VEL
LIN {X 0,Y 433.115,Z 397.388,A -85,B 0,C 180,E1 -9263.595,E2 -9263.595} C_VEL
LIN {X 0,Y 433.463,Z 389.329,A -85,B 0,C 180,E1 -9264.301,E2 -9264.301} C_VEL
LIN {X 0,Y 433.794,Z 380.972,A -85,B 0,C 180,E1 -9264.888,E2 -9264.888} C_VEL
LIN {X 0,Y 433.976,Z 372.526,A -85,B 0,C 180,E1 -9265.356,E2 -9265.356} C_VEL
LIN {X 0,Y 434.191,Z 362.455,A -85,B 0,C 180,E1 -9265.765,E2 -9265.765} C_VEL
LIN {X 0,Y 434.382,Z 350.989,A -85,B 0,C 180,E1 -9266.057,E2 -9266.057} C_VEL
LIN {X 0,Y 434.713,Z 292.124,A -85,B 0,C 180,E1 -9267.032,E2 -9267.032} C_VEL
LIN {X 0,Y 432.381,Z 279.304,A -85,B 0,C 180,E1 -9267.322,E2 -9267.322} C_VEL
LIN {X 0,Y 432.681,Z 268.541,A -85,B 0,C 180,E1 -9270,E2 -9270} C_VEL
LIN {X 0,Y 432.547,Z 266.42,A -85,B 0,C 180,E1 -9270.582,E2 -9270.582} C_VEL
LIN {X 0,Y 432.568,Z 266.414,A -85,B 0,C 180,E1 -9272.794,E2 -9272.794} C_VEL
LIN {X 0,Y 432.533,Z 266.416,A -85,B 0,C 180,E1 -9276.531,E2 -9276.531} C_VEL
LIN {X 0,Y 432.406,Z 266.437,A -85,B 0,C 180,E1 -9279.354,E2 -9279.354} C_VEL
LIN {X 0,Y 432.394,Z 266.434,A -85,B 0,C 180,E1 -9282.804,E2 -9282.804} C_VEL
LIN {X 0,Y 432.377,Z 266.435,A -85,B 0,C 180,E1 -9286.48,E2 -9286.48} C_VEL
LIN {X 0,Y 432.303,Z 266.445,A -85,B 0,C 180,E1 -9289.962,E2 -9289.962} C_VEL
LIN {X 0,Y 432.282,Z 266.448,A -85,B 0,C 180,E1 -9292.967,E2 -9292.967} C_VEL
LIN {X 0,Y 432.304,Z 266.446,A -85,B 0,C 180,E1 -9295.004,E2 -9295.004} C_VEL
LIN {X 0,Y 432.311,Z 266.443,A -85,B 0,C 180,E1 -9298.129,E2 -9298.129} C_VEL
LIN {X 0,Y 432.29,Z 266.451,A -85,B 0,C 180,E1 -9301.349,E2 -9301.349} C_VEL
LIN {X 0,Y 432.31,Z 266.443,A -85,B 0,C 180,E1 -9304.68,E2 -9304.68} C_VEL
LIN {X 0,Y 432.302,Z 266.445,A -85,B 0,C 180,E1 -9308.154,E2 -9308.154} C_VEL
LIN {X 0,Y 432.295,Z 266.45,A -85,B 0,C 180,E1 -9311.802,E2 -9311.802} C_VEL
LIN {X 0,Y 432.31,Z 266.444,A -85,B 0,C 180,E1 -9314.351,E2 -9314.351} C_VEL
LIN {X 0,Y 432.298,Z 266.445,A -85,B 0,C 180,E1 -9317.019,E2 -9317.019} C_VEL
LIN {X 0,Y 432.314,Z 266.449,A -85,B 0,C 180,E1 -9319.824,E2 -9319.824} C_VEL
LIN {X 0,Y 432.288,Z 266.447,A -85,B 0,C 180,E1 -9323.025,E2 -9323.025} C_VEL
LIN {X 0,Y 432.341,Z 266.444,A -85,B 0,C 180,E1 -9326.001,E2 -9326.001} C_VEL
LIN {X 0,Y 432.332,Z 266.444,A -85,B 0,C 180,E1 -9329.494,E2 -9329.494} C_VEL
LIN {X 0,Y 432.335,Z 266.447,A -85,B 0,C 180,E1 -9331.878,E2 -9331.878} C_VEL
LIN {X 0,Y 432.367,Z 266.439,A -85,B 0,C 180,E1 -9335.542,E2 -9335.542} C_VEL
LIN {X 0,Y 432.342,Z 266.44,A -85,B 0,C 180,E1 -9339.05,E2 -9339.05} C_VEL
LIN {X 0,Y 432.412,Z 266.433,A -85,B 0,C 180,E1 -9342.505,E2 -9342.505} C_VEL
LIN {X 0,Y 432.438,Z 266.517,A -85,B 0,C 180,E1 -9342.872,E2 -9342.872} C_VEL
LIN {X 0,Y 432.346,Z 276.773,A -85,B 0,C 180,E1 -9345.41,E2 -9345.41} C_VEL
LIN {X 0,Y 432.32,Z 278.855,A -85,B 0,C 180,E1 -9345.909,E2 -9345.909} C_VEL
LIN {X 0,Y 434.537,Z 293.834,A -85,B 0,C 180,E1 -9346.27,E2 -9346.27} C_VEL
LIN {X 0,Y 433.796,Z 356.722,A -85,B 0,C 180,E1 -9347.519,E2 -9347.519} C_VEL
LIN {X 0,Y 433.595,Z 366.942,A -85,B 0,C 180,E1 -9347.869,E2 -9347.869} C_VEL
LIN {X 0,Y 433.343,Z 377.146,A -85,B 0,C 180,E1 -9348.366,E2 -9348.366} C_VEL
LIN {X 0,Y 433.077,Z 388.53,A -85,B 0,C 180,E1 -9349.129,E2 -9349.129} C_VEL
LIN {X 0,Y 432.788,Z 396.639,A -85,B 0,C 180,E1 -9349.832,E2 -9349.832} C_VEL
LIN {X 0,Y 432.501,Z 404.386,A -85,B 0,C 180,E1 -9350.652,E2 -9350.652} C_VEL
LIN {X 0,Y 432.162,Z 411.67,A -85,B 0,C 180,E1 -9351.587,E2 -9351.587} C_VEL
LIN {X 0,Y 431.955,Z 419.083,A -85,B 0,C 180,E1 -9352.76,E2 -9352.76} C_VEL
LIN {X 0,Y 431.719,Z 424.846,A -85,B 0,C 180,E1 -9353.929,E2 -9353.929} C_VEL
LIN {X 0,Y 431.553,Z 428.618,A -85,B 0,C 180,E1 -9354.864,E2 -9354.864} C_VEL
LIN {X 0,Y 431.536,Z 431.683,A -85,B 0,C 180,E1 -9355.8,E2 -9355.8} C_VEL
LIN {X 0,Y 431.387,Z 435.031,A -85,B 0,C 180,E1 -9357.202,E2 -9357.202} C_VEL
LIN {X 0,Y 431.275,Z 436.619,A -85,B 0,C 180,E1 -9358.135,E2 -9358.135} C_VEL
LIN {X 0,Y 431.227,Z 437.634,A -85,B 0,C 180,E1 -9359.069,E2 -9359.069} C_VEL
LIN {X 0,Y 431.229,Z 438.06,A -85,B 0,C 180,E1 -9360.003,E2 -9360.003} C_VEL
LIN {X 0,Y 431.256,Z 437.969,A -85,B 0,C 180,E1 -9360.937,E2 -9360.937} C_VEL
LIN {X 0,Y 431.313,Z 437.372,A -85,B 0,C 180,E1 -9361.87,E2 -9361.87} C_VEL
LIN {X 0,Y 431.415,Z 436.26,A -85,B 0,C 180,E1 -9362.804,E2 -9362.804} C_VEL
LIN {X 0,Y 431.639,Z 433.484,A -85,B 0,C 180,E1 -9364.205,E2 -9364.205} C_VEL
LIN {X 0,Y 431.717,Z 430.922,A -85,B 0,C 180,E1 -9365.14,E2 -9365.14} C_VEL
LIN {X 0,Y 431.819,Z 427.718,A -85,B 0,C 180,E1 -9366.075,E2 -9366.075} C_VEL
LIN {X 0,Y 432.137,Z 422.748,A -85,B 0,C 180,E1 -9367.221,E2 -9367.221} C_VEL
LIN {X 0,Y 432.345,Z 417.646,A -85,B 0,C 180,E1 -9368.18,E2 -9368.18} C_VEL
LIN {X 0,Y 432.679,Z 411.619,A -85,B 0,C 180,E1 -9369.115,E2 -9369.115} C_VEL
LIN {X 0,Y 433.094,Z 404.306,A -85,B 0,C 180,E1 -9370.049,E2 -9370.049} C_VEL
LIN {X 0,Y 433.519,Z 395.296,A -85,B 0,C 180,E1 -9370.984,E2 -9370.984} C_VEL
LIN {X 0,Y 433.959,Z 384.986,A -85,B 0,C 180,E1 -9371.801,E2 -9371.801} C_VEL
LIN {X 0,Y 434.272,Z 375.549,A -85,B 0,C 180,E1 -9372.385,E2 -9372.385} C_VEL
LIN {X 0,Y 434.551,Z 364.092,A -85,B 0,C 180,E1 -9372.911,E2 -9372.911} C_VEL
LIN {X 0,Y 434.856,Z 351.747,A -85,B 0,C 180,E1 -9373.252,E2 -9373.252} C_VEL
LIN {X 0,Y 435.756,Z 293.534,A -85,B 0,C 180,E1 -9374.476,E2 -9374.476} C_VEL
LIN {X 0,Y 432.961,Z 280.439,A -85,B 0,C 180,E1 -9374.922,E2 -9374.922} C_VEL
LIN {X 0,Y 433.103,Z 270.862,A -85,B 0,C 180,E1 -9377.229,E2 -9377.229} C_VEL
LIN {X 0,Y 432.407,Z 266.445,A -85,B 0,C 180,E1 -9378.358,E2 -9378.358} C_VEL
LIN {X 0,Y 432.353,Z 266.444,A -85,B 0,C 180,E1 -9382.096,E2 -9382.096} C_VEL
LIN {X 0,Y 432.343,Z 266.444,A -85,B 0,C 180,E1 -9385.004,E2 -9385.004} C_VEL
LIN {X 0,Y 432.355,Z 266.442,A -85,B 0,C 180,E1 -9388.127,E2 -9388.127} C_VEL
LIN {X 0,Y 432.329,Z 266.443,A -85,B 0,C 180,E1 -9391.348,E2 -9391.348} C_VEL
LIN {X 0,Y 432.336,Z 266.446,A -85,B 0,C 180,E1 -9394.68,E2 -9394.68} C_VEL
LIN {X 0,Y 432.338,Z 266.445,A -85,B 0,C 180,E1 -9398.152,E2 -9398.152} C_VEL
LIN {X 0,Y 432.329,Z 266.443,A -85,B 0,C 180,E1 -9401.8,E2 -9401.8} C_VEL
LIN {X 0,Y 432.343,Z 266.444,A -85,B 0,C 180,E1 -9404.348,E2 -9404.348} C_VEL
LIN {X 0,Y 432.325,Z 266.443,A -85,B 0,C 180,E1 -9407.017,E2 -9407.017} C_VEL
LIN {X 0,Y 432.322,Z 266.443,A -85,B 0,C 180,E1 -9409.825,E2 -9409.825} C_VEL
LIN {X 0,Y 432.312,Z 266.443,A -85,B 0,C 180,E1 -9413.022,E2 -9413.022} C_VEL
LIN {X 0,Y 432.341,Z 266.44,A -85,B 0,C 180,E1 -9416.003,E2 -9416.003} C_VEL
LIN {X 0,Y 432.355,Z 266.44,A -85,B 0,C 180,E1 -9419.49,E2 -9419.49} C_VEL
LIN {X 0,Y 432.398,Z 266.436,A -85,B 0,C 180,E1 -9422.928,E2 -9422.928} C_VEL
LIN {X 0,Y 432.43,Z 266.451,A -85,B 0,C 180,E1 -9425.072,E2 -9425.072} C_VEL
LIN {X 0,Y 433.892,Z 275.768,A -85,B 0,C 180,E1 -9427.124,E2 -9427.124} C_VEL
LIN {X 0,Y 433.263,Z 290.464,A -85,B 0,C 180,E1 -9430.193,E2 -9430.193} C_VEL
LIN {X 0,Y 432.511,Z 307.044,A -85,B 0,C 180,E1 -9433.614,E2 -9433.614} C_VEL
LIN {X 0,Y 432.221,Z 315.502,A -85,B 0,C 180,E1 -9435.351,E2 -9435.351} C_VEL
LIN {X 0,Y 434.308,Z 332.811,A -85,B 0,C 180,E1 -9435.845,E2 -9435.845} C_VEL
LIN {X 0,Y 434.844,Z 341.173,A -85,B 0,C 180,E1 -9436.056,E2 -9436.056} C_VEL
LIN {X 0,Y 434.448,Z 367.732,A -85,B 0,C 180,E1 -9436.6,E2 -9436.6} C_VEL
LIN {X 0,Y 434.211,Z 395.168,A -85,B 0,C 180,E1 -9437.081,E2 -9437.081} C_VEL
LIN {X 0,Y 433.906,Z 405.632,A -85,B 0,C 180,E1 -9437.399,E2 -9437.399} C_VEL
LIN {X 0,Y 433.457,Z 417.337,A -85,B 0,C 180,E1 -9437.951,E2 -9437.951} C_VEL
LIN {X 0,Y 433.078,Z 426.267,A -85,B 0,C 180,E1 -9438.533,E2 -9438.533} C_VEL
LIN {X 0,Y 432.719,Z 434.757,A -85,B 0,C 180,E1 -9439.235,E2 -9439.235} C_VEL
LIN {X 0,Y 432.342,Z 442.766,A -85,B 0,C 180,E1 -9440.054,E2 -9440.054} C_VEL
LIN {X 0,Y 432.043,Z 449.383,A -85,B 0,C 180,E1 -9440.874,E2 -9440.874} C_VEL
LIN {X 0,Y 431.746,Z 455.669,A -85,B 0,C 180,E1 -9441.811,E2 -9441.811} C_VEL
LIN {X 0,Y 431.616,Z 460.893,A -85,B 0,C 180,E1 -9442.75,E2 -9442.75} C_VEL
LIN {X 0,Y 431.382,Z 464.979,A -85,B 0,C 180,E1 -9443.625,E2 -9443.625} C_VEL
LIN {X 0,Y 431.35,Z 469.608,A -85,B 0,C 180,E1 -9444.859,E2 -9444.859} C_VEL
LIN {X 0,Y 431.243,Z 472.38,A -85,B 0,C 180,E1 -9445.794,E2 -9445.794} C_VEL
LIN {X 0,Y 431.316,Z 475.406,A -85,B 0,C 180,E1 -9447.198,E2 -9447.198} C_VEL
LIN {X 0,Y 431.244,Z 476.754,A -85,B 0,C 180,E1 -9448.132,E2 -9448.132} C_VEL
LIN {X 0,Y 431.222,Z 477.623,A -85,B 0,C 180,E1 -9449.066,E2 -9449.066} C_VEL
LIN {X 0,Y 431.225,Z 477.937,A -85,B 0,C 180,E1 -9450,E2 -9450} C_VEL
LIN {X 0,Y 431.209,Z 477.694,A -85,B 0,C 180,E1 -9450.934,E2 -9450.934} C_VEL
LIN {X 0,Y 431.244,Z 476.99,A -85,B 0,C 180,E1 -9451.868,E2 -9451.868} C_VEL
LIN {X 0,Y 431.297,Z 475.812,A -85,B 0,C 180,E1 -9452.802,E2 -9452.802} C_VEL
LIN {X 0,Y 431.242,Z 472.971,A -85,B 0,C 180,E1 -9454.205,E2 -9454.205} C_VEL
LIN {X 0,Y 431.335,Z 468.874,A -85,B 0,C 180,E1 -9455.61,E2 -9455.61} C_VEL
LIN {X 0,Y 431.615,Z 463.355,A -85,B 0,C 180,E1 -9457.014,E2 -9457.014} C_VEL
LIN {X 0,Y 431.79,Z 457.312,A -85,B 0,C 180,E1 -9458.188,E2 -9458.188} C_VEL
LIN {X 0,Y 432.117,Z 451.424,A -85,B 0,C 180,E1 -9459.124,E2 -9459.124} C_VEL
LIN {X 0,Y 432.532,Z 444.268,A -85,B 0,C 180,E1 -9460.059,E2 -9460.059} C_VEL
LIN {X 0,Y 432.955,Z 436.652,A -85,B 0,C 180,E1 -9460.877,E2 -9460.877} C_VEL
LIN {X 0,Y 433.349,Z 428.682,A -85,B 0,C 180,E1 -9461.577,E2 -9461.577} C_VEL
LIN {X 0,Y 433.726,Z 420.468,A -85,B 0,C 180,E1 -9462.16,E2 -9462.16} C_VEL
LIN {X 0,Y 434.102,Z 412.16,A -85,B 0,C 180,E1 -9462.624,E2 -9462.624} C_VEL
LIN {X 0,Y 434.45,Z 403.207,A -85,B 0,C 180,E1 -9463,E2 -9463} C_VEL
LIN {X 0,Y 434.789,Z 394.198,A -85,B 0,C 180,E1 -9463.258,E2 -9463.258} C_VEL
LIN {X 0,Y 435.142,Z 338.068,A -85,B 0,C 180,E1 -9464.223,E2 -9464.223} C_VEL
LIN {X 0,Y 432.672,Z 319.011,A -85,B 0,C 180,E1 -9464.644,E2 -9464.644} C_VEL
LIN {X 0,Y 432.347,Z 316.664,A -85,B 0,C 180,E1 -9464.711,E2 -9464.711} C_VEL
LIN {X 0,Y 432.915,Z 302.091,A -85,B 0,C 180,E1 -9467.721,E2 -9467.721} C_VEL
LIN {X 0,Y 433.667,Z 286.929,A -85,B 0,C 180,E1 -9470.887,E2 -9470.887} C_VEL
LIN {X 0,Y 434.153,Z 276.432,A -85,B 0,C 180,E1 -9473.113,E2 -9473.113} C_VEL
LIN {X 0,Y 432.389,Z 266.442,A -85,B 0,C 180,E1 -9475.417,E2 -9475.417} C_VEL
LIN {X 0,Y 432.381,Z 266.438,A -85,B 0,C 180,E1 -9478.628,E2 -9478.628} C_VEL
LIN {X 0,Y 432.325,Z 266.447,A -85,B 0,C 180,E1 -9481.346,E2 -9481.346} C_VEL
LIN {X 0,Y 432.334,Z 266.444,A -85,B 0,C 180,E1 -9484.677,E2 -9484.677} C_VEL
LIN {X 0,Y 432.337,Z 266.441,A -85,B 0,C 180,E1 -9488.15,E2 -9488.15} C_VEL
LIN {X 0,Y 432.332,Z 266.445,A -85,B 0,C 180,E1 -9491.6,E2 -9491.6} C_VEL
LIN {X 0,Y 432.341,Z 266.438,A -85,B 0,C 180,E1 -9494.346,E2 -9494.346} C_VEL
LIN {X 0,Y 432.324,Z 266.444,A -85,B 0,C 180,E1 -9497.015,E2 -9497.015} C_VEL
LIN {X 0,Y 432.321,Z 266.444,A -85,B 0,C 180,E1 -9499.823,E2 -9499.823} C_VEL
LIN {X 0,Y 432.312,Z 266.444,A -85,B 0,C 180,E1 -9503.02,E2 -9503.02} C_VEL
LIN {X 0,Y 432.364,Z 266.44,A -85,B 0,C 180,E1 -9505.995,E2 -9505.995} C_VEL
LIN {X 0,Y 432.353,Z 266.438,A -85,B 0,C 180,E1 -9509.488,E2 -9509.488} C_VEL
LIN {X 0,Y 432.35,Z 266.442,A -85,B 0,C 180,E1 -9511.872,E2 -9511.872} C_VEL
LIN {X 0,Y 432.385,Z 266.437,A -85,B 0,C 180,E1 -9515.536,E2 -9515.536} C_VEL
LIN {X 0,Y 432.356,Z 266.432,A -85,B 0,C 180,E1 -9519.044,E2 -9519.044} C_VEL
LIN {X 0,Y 432.365,Z 266.438,A -85,B 0,C 180,E1 -9522.008,E2 -9522.008} C_VEL
LIN {X 0,Y 432.399,Z 266.428,A -85,B 0,C 180,E1 -9524.924,E2 -9524.924} C_VEL
LIN {X 0,Y 432.463,Z 266.426,A -85,B 0,C 180,E1 -9527.801,E2 -9527.801} C_VEL
LIN {X 0,Y 432.495,Z 266.42,A -85,B 0,C 180,E1 -9531.588,E2 -9531.588} C_VEL
LIN {X 0,Y 432.596,Z 266.403,A -85,B 0,C 180,E1 -9534.403,E2 -9534.403} C_VEL
LIN {X 0,Y 432.601,Z 266.408,A -85,B 0,C 180,E1 -9538.135,E2 -9538.135} C_VEL
LIN {X 0,Y 432.728,Z 266.389,A -85,B 0,C 180,E1 -9539.997,E2 -9539.997} C_VEL
LIN {X 0,Y 432.583,Z 266.408,A -85,B 0,C 180,E1 -9542.791,E2 -9542.791} C_VEL
LIN {X 0,Y 432.581,Z 266.403,A -85,B 0,C 180,E1 -9545.591,E2 -9545.591} C_VEL
LIN {X 0,Y 432.46,Z 266.428,A -85,B 0,C 180,E1 -9548.407,E2 -9548.407} C_VEL
LIN {X 0,Y 432.454,Z 266.429,A -85,B 0,C 180,E1 -9552.193,E2 -9552.193} C_VEL
LIN {X 0,Y 432.423,Z 266.428,A -85,B 0,C 180,E1 -9556.035,E2 -9556.035} C_VEL
LIN {X 0,Y 432.377,Z 266.433,A -85,B 0,C 180,E1 -9559.482,E2 -9559.482} C_VEL
LIN {X 0,Y 432.308,Z 266.444,A -85,B 0,C 180,E1 -9562.961,E2 -9562.961} C_VEL
LIN {X 0,Y 432.351,Z 266.44,A -85,B 0,C 180,E1 -9566.029,E2 -9566.029} C_VEL
LIN {X 0,Y 432.328,Z 266.442,A -85,B 0,C 180,E1 -9569.184,E2 -9569.184} C_VEL
LIN {X 0,Y 432.306,Z 266.448,A -85,B 0,C 180,E1 -9572.439,E2 -9572.439} C_VEL
LIN {X 0,Y 432.326,Z 266.434,A -85,B 0,C 180,E1 -9575.629,E2 -9575.629} C_VEL
LIN {X 0,Y 432.325,Z 266.44,A -85,B 0,C 180,E1 -9579.34,E2 -9579.34} C_VEL
LIN {X 0,Y 432.348,Z 266.44,A -85,B 0,C 180,E1 -9581.789,E2 -9581.789} C_VEL
LIN {X 0,Y 432.355,Z 266.439,A -85,B 0,C 180,E1 -9584.338,E2 -9584.338} C_VEL
LIN {X 0,Y 432.341,Z 266.442,A -85,B 0,C 180,E1 -9587.006,E2 -9587.006} C_VEL
LIN {X 0,Y 432.332,Z 266.443,A -85,B 0,C 180,E1 -9589.814,E2 -9589.814} C_VEL
LIN {X 0,Y 432.289,Z 266.453,A -85,B 0,C 180,E1 -9593.02,E2 -9593.02} C_VEL
LIN {X 0,Y 432.354,Z 266.574,A -85,B 0,C 180,E1 -9595.218,E2 -9595.218} C_VEL
LIN {X 0,Y 432.894,Z 270.467,A -85,B 0,C 180,E1 -9596.201,E2 -9596.201} C_VEL
LIN {X 0,Y 432.751,Z 279.553,A -85,B 0,C 180,E1 -9598.366,E2 -9598.366} C_VEL
LIN {X 0,Y 435.608,Z 294.357,A -85,B 0,C 180,E1 -9598.735,E2 -9598.735} C_VEL
LIN {X 0,Y 434.942,Z 356.257,A -85,B 0,C 180,E1 -9599.794,E2 -9599.794} C_VEL
LIN {X 0,Y 434.756,Z 366.912,A -85,B 0,C 180,E1 -9600.126,E2 -9600.126} C_VEL
LIN {X 0,Y 434.432,Z 379.113,A -85,B 0,C 180,E1 -9600.728,E2 -9600.728} C_VEL
LIN {X 0,Y 434.06,Z 388.094,A -85,B 0,C 180,E1 -9601.336,E2 -9601.336} C_VEL
LIN {X 0,Y 433.722,Z 395.612,A -85,B 0,C 180,E1 -9601.971,E2 -9601.971} C_VEL
LIN {X 0,Y 433.255,Z 402.978,A -85,B 0,C 180,E1 -9602.726,E2 -9602.726} C_VEL
LIN {X 0,Y 432.875,Z 409.554,A -85,B 0,C 180,E1 -9603.54,E2 -9603.54} C_VEL
LIN {X 0,Y 432.511,Z 415.932,A -85,B 0,C 180,E1 -9604.494,E2 -9604.494} C_VEL
LIN {X 0,Y 432.256,Z 420.692,A -85,B 0,C 180,E1 -9605.344,E2 -9605.344} C_VEL
LIN {X 0,Y 431.922,Z 426.022,A -85,B 0,C 180,E1 -9606.506,E2 -9606.506} C_VEL
LIN {X 0,Y 431.685,Z 429.714,A -85,B 0,C 180,E1 -9607.506,E2 -9607.506} C_VEL
LIN {X 0,Y 431.541,Z 432.828,A -85,B 0,C 180,E1 -9608.57,E2 -9608.57} C_VEL
LIN {X 0,Y 431.343,Z 435.811,A -85,B 0,C 180,E1 -9609.992,E2 -9609.992} C_VEL
LIN {X 0,Y 431.263,Z 437.167,A -85,B 0,C 180,E1 -9610.978,E2 -9610.978} C_VEL
LIN {X 0,Y 431.2,Z 437.982,A -85,B 0,C 180,E1 -9611.96,E2 -9611.96} C_VEL
LIN {X 0,Y 431.166,Z 438.263,A -85,B 0,C 180,E1 -9612.939,E2 -9612.939} C_VEL
LIN {X 0,Y 431.213,Z 437.871,A -85,B 0,C 180,E1 -9614.051,E2 -9614.051} C_VEL
LIN {X 0,Y 431.236,Z 437.052,A -85,B 0,C 180,E1 -9614.885,E2 -9614.885} C_VEL
LIN {X 0,Y 431.275,Z 435.659,A -85,B 0,C 180,E1 -9615.852,E2 -9615.852} C_VEL
LIN {X 0,Y 431.439,Z 432.54,A -85,B 0,C 180,E1 -9617.297,E2 -9617.297} C_VEL
LIN {X 0,Y 431.644,Z 428.077,A -85,B 0,C 180,E1 -9618.733,E2 -9618.733} C_VEL
LIN {X 0,Y 431.816,Z 424.689,A -85,B 0,C 180,E1 -9619.566,E2 -9619.566} C_VEL
LIN {X 0,Y 431.328,Z 421.739,A -85,B 0,C 180,E1 -9620.243,E2 -9620.243} C_VEL
LIN {X 0,Y 428.771,Z 416.35,A -85,B 0,C 180,E1 -9621.3,E2 -9621.3} C_VEL
LIN {X 0,Y 426.203,Z 410.142,A -85,B 0,C 180,E1 -9622.283,E2 -9622.283} C_VEL
LIN {X 0,Y 425.702,Z 405.904,A -85,B 0,C 180,E1 -9622.836,E2 -9622.836} C_VEL
LIN {X 0,Y 426.106,Z 397.798,A -85,B 0,C 180,E1 -9623.727,E2 -9623.727} C_VEL
LIN {X 0,Y 426.48,Z 389.746,A -85,B 0,C 180,E1 -9624.444,E2 -9624.444} C_VEL
LIN {X 0,Y 426.812,Z 381.413,A -85,B 0,C 180,E1 -9625.041,E2 -9625.041} C_VEL
LIN {X 0,Y 427.013,Z 372.988,A -85,B 0,C 180,E1 -9625.516,E2 -9625.516} C_VEL
LIN {X 0,Y 427.226,Z 363.789,A -85,B 0,C 180,E1 -9625.903,E2 -9625.903} C_VEL
LIN {X 0,Y 427.398,Z 354.269,A -85,B 0,C 180,E1 -9626.17,E2 -9626.17} C_VEL
LIN {X 0,Y 427.76,Z 292.853,A -85,B 0,C 180,E1 -9627.223,E2 -9627.223} C_VEL
LIN {X 0,Y 425.393,Z 279.518,A -85,B 0,C 180,E1 -9627.544,E2 -9627.544} C_VEL
LIN {X 0,Y 425.672,Z 269.731,A -85,B 0,C 180,E1 -9630,E2 -9630} C_VEL
LIN {X 0,Y 425.512,Z 267.296,A -85,B 0,C 180,E1 -9630.651,E2 -9630.651} C_VEL
LIN {X 0,Y 425.52,Z 267.292,A -85,B 0,C 180,E1 -9632.84,E2 -9632.84} C_VEL
LIN {X 0,Y 425.491,Z 267.294,A -85,B 0,C 180,E1 -9636.64,E2 -9636.64} C_VEL
LIN {X 0,Y 425.365,Z 267.313,A -85,B 0,C 180,E1 -9639.51,E2 -9639.51} C_VEL
LIN {X 0,Y 425.357,Z 267.312,A -85,B 0,C 180,E1 -9642.905,E2 -9642.905} C_VEL
LIN {X 0,Y 425.326,Z 267.313,A -85,B 0,C 180,E1 -9646.606,E2 -9646.606} C_VEL
LIN {X 0,Y 425.294,Z 267.321,A -85,B 0,C 180,E1 -9649.637,E2 -9649.637} C_VEL
LIN {X 0,Y 425.269,Z 267.327,A -85,B 0,C 180,E1 -9653.368,E2 -9653.368} C_VEL
LIN {X 0,Y 425.268,Z 267.32,A -85,B 0,C 180,E1 -9656.501,E2 -9656.501} C_VEL
LIN {X 0,Y 425.254,Z 267.326,A -85,B 0,C 180,E1 -9659.723,E2 -9659.723} C_VEL
LIN {X 0,Y 425.253,Z 267.324,A -85,B 0,C 180,E1 -9663.051,E2 -9663.051} C_VEL
LIN {X 0,Y 425.253,Z 267.325,A -85,B 0,C 180,E1 -9665.931,E2 -9665.931} C_VEL
LIN {X 0,Y 425.235,Z 267.326,A -85,B 0,C 180,E1 -9669.04,E2 -9669.04} C_VEL
LIN {X 0,Y 425.245,Z 267.323,A -85,B 0,C 180,E1 -9672.657,E2 -9672.657} C_VEL
LIN {X 0,Y 425.239,Z 267.327,A -85,B 0,C 180,E1 -9676.047,E2 -9676.047} C_VEL
LIN {X 0,Y 425.253,Z 267.322,A -85,B 0,C 180,E1 -9678.625,E2 -9678.625} C_VEL
LIN {X 0,Y 425.273,Z 267.321,A -85,B 0,C 180,E1 -9681.104,E2 -9681.104} C_VEL
LIN {X 0,Y 425.281,Z 267.319,A -85,B 0,C 180,E1 -9684.668,E2 -9684.668} C_VEL
LIN {X 0,Y 425.249,Z 267.327,A -85,B 0,C 180,E1 -9688.077,E2 -9688.077} C_VEL
LIN {X 0,Y 425.301,Z 267.318,A -85,B 0,C 180,E1 -9691.37,E2 -9691.37} C_VEL
LIN {X 0,Y 425.259,Z 267.323,A -85,B 0,C 180,E1 -9694.557,E2 -9694.557} C_VEL
LIN {X 0,Y 425.274,Z 267.321,A -85,B 0,C 180,E1 -9696.637,E2 -9696.637} C_VEL
LIN {X 0,Y 425.288,Z 267.322,A -85,B 0,C 180,E1 -9699.698,E2 -9699.698} C_VEL
LIN {X 0,Y 425.385,Z 267.431,A -85,B 0,C 180,E1 -9702.851,E2 -9702.851} C_VEL
LIN {X 0,Y 425.314,Z 276.752,A -85,B 0,C 180,E1 -9705.163,E2 -9705.163} C_VEL
LIN {X 0,Y 425.281,Z 279.07,A -85,B 0,C 180,E1 -9705.724,E2 -9705.724} C_VEL
LIN {X 0,Y 427.574,Z 294.737,A -85,B 0,C 180,E1 -9706.107,E2 -9706.107} C_VEL
LIN {X 0,Y 426.799,Z 356.622,A -85,B 0,C 180,E1 -9707.371,E2 -9707.371} C_VEL
LIN {X 0,Y 426.577,Z 366.909,A -85,B 0,C 180,E1 -9707.727,E2 -9707.727} C_VEL
LIN {X 0,Y 426.337,Z 377.169,A -85,B 0,C 180,E1 -9708.233,E2 -9708.233} C_VEL
LIN {X 0,Y 426.098,Z 387.926,A -85,B 0,C 180,E1 -9708.949,E2 -9708.949} C_VEL
LIN {X 0,Y 425.739,Z 397.373,A -85,B 0,C 180,E1 -9709.782,E2 -9709.782} C_VEL
LIN {X 0,Y 425.469,Z 404.053,A -85,B 0,C 180,E1 -9710.496,E2 -9710.496} C_VEL
LIN {X 0,Y 425.126,Z 411.44,A -85,B 0,C 180,E1 -9711.447,E2 -9711.447} C_VEL
LIN {X 0,Y 424.878,Z 417.54,A -85,B 0,C 180,E1 -9712.399,E2 -9712.399} C_VEL
LIN {X 0,Y 424.699,Z 423.785,A -85,B 0,C 180,E1 -9713.59,E2 -9713.59} C_VEL
LIN {X 0,Y 424.491,Z 428.688,A -85,B 0,C 180,E1 -9714.779,E2 -9714.779} C_VEL
LIN {X 0,Y 424.386,Z 433.037,A -85,B 0,C 180,E1 -9716.205,E2 -9716.205} C_VEL
LIN {X 0,Y 424.322,Z 435.23,A -85,B 0,C 180,E1 -9717.155,E2 -9717.155} C_VEL
LIN {X 0,Y 424.2,Z 436.865,A -85,B 0,C 180,E1 -9718.104,E2 -9718.104} C_VEL
LIN {X 0,Y 424.144,Z 437.903,A -85,B 0,C 180,E1 -9719.054,E2 -9719.054} C_VEL
LIN {X 0,Y 424.143,Z 438.368,A -85,B 0,C 180,E1 -9720.003,E2 -9720.003} C_VEL
LIN {X 0,Y 424.172,Z 438.323,A -85,B 0,C 180,E1 -9720.952,E2 -9720.952} C_VEL
LIN {X 0,Y 424.236,Z 437.769,A -85,B 0,C 180,E1 -9721.902,E2 -9721.902} C_VEL
LIN {X 0,Y 424.35,Z 436.697,A -85,B 0,C 180,E1 -9722.851,E2 -9722.851} C_VEL
LIN {X 0,Y 424.593,Z 433.954,A -85,B 0,C 180,E1 -9724.275,E2 -9724.275} C_VEL
LIN {X 0,Y 424.67,Z 431.429,A -85,B 0,C 180,E1 -9725.225,E2 -9725.225} C_VEL
LIN {X 0,Y 424.793,Z 428.258,A -85,B 0,C 180,E1 -9726.176,E2 -9726.176} C_VEL
LIN {X 0,Y 425.13,Z 423.501,A -85,B 0,C 180,E1 -9727.302,E2 -9727.302} C_VEL
LIN {X 0,Y 425.367,Z 418.258,A -85,B 0,C 180,E1 -9728.315,E2 -9728.315} C_VEL
LIN {X 0,Y 425.723,Z 412.309,A -85,B 0,C 180,E1 -9729.265,E2 -9729.265} C_VEL
LIN {X 0,Y 426.151,Z 405.095,A -85,B 0,C 180,E1 -9730.214,E2 -9730.214} C_VEL
LIN {X 0,Y 426.614,Z 396.24,A -85,B 0,C 180,E1 -9731.164,E2 -9731.164} C_VEL
LIN {X 0,Y 427.117,Z 386.166,A -85,B 0,C 180,E1 -9731.992,E2 -9731.992} C_VEL
LIN {X 0,Y 427.435,Z 376.929,A -85,B 0,C 180,E1 -9732.586,E2 -9732.586} C_VEL
LIN {X 0,Y 427.689,Z 367.229,A -85,B 0,C 180,E1 -9733.061,E2 -9733.061} C_VEL
LIN {X 0,Y 427.988,Z 355.389,A -85,B 0,C 180,E1 -9733.454,E2 -9733.454} C_VEL
LIN {X 0,Y 429.085,Z 294.442,A -85,B 0,C 180,E1 -9734.777,E2 -9734.777} C_VEL
LIN {X 0,Y 426.056,Z 280.698,A -85,B 0,C 180,E1 -9735.274,E2 -9735.274} C_VEL
LIN {X 0,Y 426.115,Z 271.524,A -85,B 0,C 180,E1 -9737.52,E2 -9737.52} C_VEL
LIN {X 0,Y 425.357,Z 267.322,A -85,B 0,C 180,E1 -9738.611,E2 -9738.611} C_VEL
LIN {X 0,Y 425.296,Z 267.323,A -85,B 0,C 180,E1 -9742.341,E2 -9742.341} C_VEL
LIN {X 0,Y 425.326,Z 267.319,A -85,B 0,C 180,E1 -9744.658,E2 -9744.658} C_VEL
LIN {X 0,Y 425.279,Z 267.323,A -85,B 0,C 180,E1 -9747.565,E2 -9747.565} C_VEL
LIN {X 0,Y 425.299,Z 267.322,A -85,B 0,C 180,E1 -9750.762,E2 -9750.762} C_VEL
LIN {X 0,Y 425.3,Z 267.322,A -85,B 0,C 180,E1 -9754.285,E2 -9754.285} C_VEL
LIN {X 0,Y 425.284,Z 267.321,A -85,B 0,C 180,E1 -9757.696,E2 -9757.696} C_VEL
LIN {X 0,Y 425.255,Z 267.328,A -85,B 0,C 180,E1 -9760.516,E2 -9760.516} C_VEL
LIN {X 0,Y 425.264,Z 267.321,A -85,B 0,C 180,E1 -9763.351,E2 -9763.351} C_VEL
LIN {X 0,Y 425.27,Z 267.322,A -85,B 0,C 180,E1 -9766.045,E2 -9766.045} C_VEL
LIN {X 0,Y 425.273,Z 267.324,A -85,B 0,C 180,E1 -9768.621,E2 -9768.621} C_VEL
LIN {X 0,Y 425.289,Z 267.321,A -85,B 0,C 180,E1 -9771.1,E2 -9771.1} C_VEL
LIN {X 0,Y 425.303,Z 267.322,A -85,B 0,C 180,E1 -9774.664,E2 -9774.664} C_VEL
LIN {X 0,Y 425.271,Z 267.323,A -85,B 0,C 180,E1 -9778.073,E2 -9778.073} C_VEL
LIN {X 0,Y 425.339,Z 267.315,A -85,B 0,C 180,E1 -9781.368,E2 -9781.368} C_VEL
LIN {X 0,Y 425.391,Z 267.313,A -85,B 0,C 180,E1 -9784.936,E2 -9784.936} C_VEL
LIN {X 0,Y 426.903,Z 276.675,A -85,B 0,C 180,E1 -9787.035,E2 -9787.035} C_VEL
LIN {X 0,Y 426.264,Z 290.724,A -85,B 0,C 180,E1 -9790.018,E2 -9790.018} C_VEL
LIN {X 0,Y 425.422,Z 308.222,A -85,B 0,C 180,E1 -9793.689,E2 -9793.689} C_VEL
LIN {X 0,Y 425.231,Z 314.437,A -85,B 0,C 180,E1 -9794.987,E2 -9794.987} C_VEL
LIN {X 0,Y 427.275,Z 330.533,A -85,B 0,C 180,E1 -9795.474,E2 -9795.474} C_VEL
LIN {X 0,Y 428.099,Z 341.64,A -85,B 0,C 180,E1 -9795.769,E2 -9795.769} C_VEL
LIN {X 0,Y 427.382,Z 387.563,A -85,B 0,C 180,E1 -9796.75,E2 -9796.75} C_VEL
LIN {X 0,Y 427.121,Z 400.288,A -85,B 0,C 180,E1 -9797.045,E2 -9797.045} C_VEL
LIN {X 0,Y 426.738,Z 410.668,A -85,B 0,C 180,E1 -9797.456,E2 -9797.456} C_VEL
LIN {X 0,Y 426.414,Z 418.396,A -85,B 0,C 180,E1 -9797.869,E2 -9797.869} C_VEL
LIN {X 0,Y 426.052,Z 427.056,A -85,B 0,C 180,E1 -9798.462,E2 -9798.462} C_VEL
LIN {X 0,Y 425.669,Z 435.344,A -85,B 0,C 180,E1 -9799.175,E2 -9799.175} C_VEL
LIN {X 0,Y 425.262,Z 443.197,A -85,B 0,C 180,E1 -9800.007,E2 -9800.007} C_VEL
LIN {X 0,Y 424.931,Z 450.55,A -85,B 0,C 180,E1 -9800.96,E2 -9800.96} C_VEL
LIN {X 0,Y 424.597,Z 457.998,A -85,B 0,C 180,E1 -9802.151,E2 -9802.151} C_VEL
LIN {X 0,Y 424.359,Z 463.816,A -85,B 0,C 180,E1 -9803.343,E2 -9803.343} C_VEL
LIN {X 0,Y 424.241,Z 467.63,A -85,B 0,C 180,E1 -9804.295,E2 -9804.295} C_VEL
LIN {X 0,Y 424.166,Z 471.979,A -85,B 0,C 180,E1 -9805.724,E2 -9805.724} C_VEL
LIN {X 0,Y 424.226,Z 475.027,A -85,B 0,C 180,E1 -9807.151,E2 -9807.151} C_VEL
LIN {X 0,Y 424.17,Z 476.397,A -85,B 0,C 180,E1 -9808.101,E2 -9808.101} C_VEL
LIN {X 0,Y 424.139,Z 477.284,A -85,B 0,C 180,E1 -9809.05,E2 -9809.05} C_VEL
LIN {X 0,Y 424.139,Z 477.599,A -85,B 0,C 180,E1 -9810,E2 -9810} C_VEL
LIN {X 0,Y 424.127,Z 477.377,A -85,B 0,C 180,E1 -9810.949,E2 -9810.949} C_VEL
LIN {X 0,Y 424.169,Z 476.693,A -85,B 0,C 180,E1 -9811.899,E2 -9811.899} C_VEL
LIN {X 0,Y 424.193,Z 475.534,A -85,B 0,C 180,E1 -9812.849,E2 -9812.849} C_VEL
LIN {X 0,Y 424.165,Z 472.714,A -85,B 0,C 180,E1 -9814.276,E2 -9814.276} C_VEL
LIN {X 0,Y 424.243,Z 468.638,A -85,B 0,C 180,E1 -9815.704,E2 -9815.704} C_VEL
LIN {X 0,Y 424.549,Z 463.155,A -85,B 0,C 180,E1 -9817.132,E2 -9817.132} C_VEL
LIN {X 0,Y 424.751,Z 457.167,A -85,B 0,C 180,E1 -9818.324,E2 -9818.324} C_VEL
LIN {X 0,Y 425.2,Z 449.618,A -85,B 0,C 180,E1 -9819.514,E2 -9819.514} C_VEL
LIN {X 0,Y 425.574,Z 443.202,A -85,B 0,C 180,E1 -9820.346,E2 -9820.346} C_VEL
LIN {X 0,Y 426.023,Z 435.447,A -85,B 0,C 180,E1 -9821.177,E2 -9821.177} C_VEL
LIN {X 0,Y 426.507,Z 427.298,A -85,B 0,C 180,E1 -9821.886,E2 -9821.886} C_VEL
LIN {X 0,Y 426.876,Z 418.84,A -85,B 0,C 180,E1 -9822.479,E2 -9822.479} C_VEL
LIN {X 0,Y 427.36,Z 408.964,A -85,B 0,C 180,E1 -9823.008,E2 -9823.008} C_VEL
LIN {X 0,Y 427.892,Z 397.145,A -85,B 0,C 180,E1 -9823.436,E2 -9823.436} C_VEL
LIN {X 0,Y 428.126,Z 379.737,A -85,B 0,C 180,E1 -9823.774,E2 -9823.774} C_VEL
LIN {X 0,Y 428.374,Z 339.147,A -85,B 0,C 180,E1 -9824.467,E2 -9824.467} C_VEL
LIN {X 0,Y 425.989,Z 320.603,A -85,B 0,C 180,E1 -9824.884,E2 -9824.884} C_VEL
LIN {X 0,Y 425.352,Z 316.347,A -85,B 0,C 180,E1 -9824.992,E2 -9824.992} C_VEL
LIN {X 0,Y 426.086,Z 299.613,A -85,B 0,C 180,E1 -9828.513,E2 -9828.513} C_VEL
LIN {X 0,Y 426.838,Z 285.639,A -85,B 0,C 180,E1 -9831.491,E2 -9831.491} C_VEL
LIN {X 0,Y 427.186,Z 277.474,A -85,B 0,C 180,E1 -9833.256,E2 -9833.256} C_VEL
LIN {X 0,Y 425.343,Z 267.319,A -85,B 0,C 180,E1 -9835.639,E2 -9835.639} C_VEL
LIN {X 0,Y 425.336,Z 267.318,A -85,B 0,C 180,E1 -9838.865,E2 -9838.865} C_VEL
LIN {X 0,Y 425.269,Z 267.319,A -85,B 0,C 180,E1 -9841.926,E2 -9841.926} C_VEL
LIN {X 0,Y 425.302,Z 267.316,A -85,B 0,C 180,E1 -9845.335,E2 -9845.335} C_VEL
LIN {X 0,Y 425.288,Z 267.321,A -85,B 0,C 180,E1 -9848.9,E2 -9848.9} C_VEL
LIN {X 0,Y 425.29,Z 267.321,A -85,B 0,C 180,E1 -9851.956,E2 -9851.956} C_VEL
LIN {X 0,Y 425.292,Z 267.321,A -85,B 0,C 180,E1 -9855.282,E2 -9855.282} C_VEL
LIN {X 0,Y 425.272,Z 267.32,A -85,B 0,C 180,E1 -9858.619,E2 -9858.619} C_VEL
LIN {X 0,Y 425.288,Z 267.318,A -85,B 0,C 180,E1 -9861.098,E2 -9861.098} C_VEL
LIN {X 0,Y 425.305,Z 267.312,A -85,B 0,C 180,E1 -9864.662,E2 -9864.662} C_VEL
LIN {X 0,Y 425.27,Z 267.319,A -85,B 0,C 180,E1 -9868.071,E2 -9868.071} C_VEL
LIN {X 0,Y 425.317,Z 267.318,A -85,B 0,C 180,E1 -9871.365,E2 -9871.365} C_VEL
LIN {X 0,Y 425.279,Z 267.318,A -85,B 0,C 180,E1 -9874.551,E2 -9874.551} C_VEL
LIN {X 0,Y 425.29,Z 267.318,A -85,B 0,C 180,E1 -9876.632,E2 -9876.632} C_VEL
LIN {X 0,Y 425.301,Z 267.316,A -85,B 0,C 180,E1 -9879.692,E2 -9879.692} C_VEL
LIN {X 0,Y 425.338,Z 267.308,A -85,B 0,C 180,E1 -9882.695,E2 -9882.695} C_VEL
LIN {X 0,Y 425.352,Z 267.311,A -85,B 0,C 180,E1 -9885.648,E2 -9885.648} C_VEL
LIN {X 0,Y 425.353,Z 267.302,A -85,B 0,C 180,E1 -9888.561,E2 -9888.561} C_VEL
LIN {X 0,Y 425.541,Z 267.285,A -85,B 0,C 180,E1 -9892.405,E2 -9892.405} C_VEL
LIN {X 0,Y 425.553,Z 267.28,A -85,B 0,C 180,E1 -9894.31,E2 -9894.31} C_VEL
LIN {X 0,Y 425.571,Z 267.284,A -85,B 0,C 180,E1 -9898.104,E2 -9898.104} C_VEL
LIN {X 0,Y 425.698,Z 267.264,A -85,B 0,C 180,E1 -9899.997,E2 -9899.997} C_VEL
LIN {X 0,Y 425.537,Z 267.285,A -85,B 0,C 180,E1 -9902.837,E2 -9902.837} C_VEL
LIN {X 0,Y 425.493,Z 267.292,A -85,B 0,C 180,E1 -9906.527,E2 -9906.527} C_VEL
LIN {X 0,Y 425.394,Z 267.303,A -85,B 0,C 180,E1 -9909.506,E2 -9909.506} C_VEL
LIN {X 0,Y 425.388,Z 267.307,A -85,B 0,C 180,E1 -9912.9,E2 -9912.9} C_VEL
LIN {X 0,Y 425.353,Z 267.313,A -85,B 0,C 180,E1 -9916.601,E2 -9916.601} C_VEL
LIN {X 0,Y 425.319,Z 267.313,A -85,B 0,C 180,E1 -9919.632,E2 -9919.632} C_VEL
LIN {X 0,Y 425.295,Z 267.316,A -85,B 0,C 180,E1 -9923.362,E2 -9923.362} C_VEL
LIN {X 0,Y 425.334,Z 267.315,A -85,B 0,C 180,E1 -9926.841,E2 -9926.841} C_VEL
LIN {X 0,Y 425.276,Z 267.32,A -85,B 0,C 180,E1 -9929.716,E2 -9929.716} C_VEL
LIN {X 0,Y 425.265,Z 267.323,A -85,B 0,C 180,E1 -9933.044,E2 -9933.044} C_VEL
LIN {X 0,Y 425.264,Z 267.315,A -85,B 0,C 180,E1 -9935.925,E2 -9935.925} C_VEL
LIN {X 0,Y 425.272,Z 267.321,A -85,B 0,C 180,E1 -9939.039,E2 -9939.039} C_VEL
LIN {X 0,Y 425.308,Z 267.323,A -85,B 0,C 180,E1 -9942.643,E2 -9942.643} C_VEL
LIN {X 0,Y 425.31,Z 267.318,A -85,B 0,C 180,E1 -9946.051,E2 -9946.051} C_VEL
LIN {X 0,Y 425.284,Z 267.324,A -85,B 0,C 180,E1 -9948.623,E2 -9948.623} C_VEL
LIN {X 0,Y 425.297,Z 267.322,A -85,B 0,C 180,E1 -9951.101,E2 -9951.101} C_VEL
LIN {X 0,Y 425.322,Z 267.451,A -85,B 0,C 180,E1 -9955.019,E2 -9955.019} C_VEL
LIN {X 0,Y 425.932,Z 271.897,A -85,B 0,C 180,E1 -9956.16,E2 -9956.16} C_VEL
LIN {X 0,Y 425.798,Z 279.607,A -85,B 0,C 180,E1 -9958.055,E2 -9958.055} C_VEL
LIN {X 0,Y 428.764,Z 294.437,A -85,B 0,C 180,E1 -9958.459,E2 -9958.459} C_VEL
LIN {X 0,Y 428.124,Z 356.103,A -85,B 0,C 180,E1 -9959.53,E2 -9959.53} C_VEL
LIN {X 0,Y 427.938,Z 366.14,A -85,B 0,C 180,E1 -9959.839,E2 -9959.839} C_VEL
LIN {X 0,Y 427.631,Z 377.896,A -85,B 0,C 180,E1 -9960.392,E2 -9960.392} C_VEL
LIN {X 0,Y 427.258,Z 387.156,A -85,B 0,C 180,E1 -9961.007,E2 -9961.007} C_VEL
LIN {X 0,Y 426.813,Z 395.866,A -85,B 0,C 180,E1 -9961.745,E2 -9961.745} C_VEL
LIN {X 0,Y 426.344,Z 403.251,A -85,B 0,C 180,E1 -9962.512,E2 -9962.512} C_VEL
LIN {X 0,Y 425.922,Z 410.004,A -85,B 0,C 180,E1 -9963.363,E2 -9963.363} C_VEL
LIN {X 0,Y 425.525,Z 416.215,A -85,B 0,C 180,E1 -9964.307,E2 -9964.307} C_VEL
LIN {X 0,Y 425.184,Z 421.956,A -85,B 0,C 180,E1 -9965.371,E2 -9965.371} C_VEL
LIN {X 0,Y 424.901,Z 426.315,A -85,B 0,C 180,E1 -9966.353,E2 -9966.353} C_VEL
LIN {X 0,Y 424.614,Z 430.814,A -85,B 0,C 180,E1 -9967.624,E2 -9967.624} C_VEL
LIN {X 0,Y 424.383,Z 434.783,A -85,B 0,C 180,E1 -9969.142,E2 -9969.142} C_VEL
LIN {X 0,Y 424.183,Z 437.373,A -85,B 0,C 180,E1 -9970.788,E2 -9970.788} C_VEL
LIN {X 0,Y 424.131,Z 438.202,A -85,B 0,C 180,E1 -9971.649,E2 -9971.649} C_VEL
LIN {X 0,Y 424.076,Z 438.548,A -85,B 0,C 180,E1 -9972.644,E2 -9972.644} C_VEL
LIN {X 0,Y 424.139,Z 438.242,A -85,B 0,C 180,E1 -9973.94,E2 -9973.94} C_VEL
LIN {X 0,Y 424.166,Z 436.425,A -85,B 0,C 180,E1 -9975.609,E2 -9975.609} C_VEL
LIN {X 0,Y 424.281,Z 434.67,A -85,B 0,C 180,E1 -9976.591,E2 -9976.591} C_VEL
LIN {X 0,Y 424.412,Z 432.033,A -85,B 0,C 180,E1 -9977.665,E2 -9977.665} C_VEL
LIN {X 0,Y 424.623,Z 427.486,A -85,B 0,C 180,E1 -9979.028,E2 -9979.028} C_VEL
LIN {X 0,Y 424.895,Z 422.25,A -85,B 0,C 180,E1 -9980.239,E2 -9980.239} C_VEL
LIN {X 0,Y 425.159,Z 417.121,A -85,B 0,C 180,E1 -9981.205,E2 -9981.205} C_VEL
LIN {X 0,Y 425.464,Z 410.762,A -85,B 0,C 180,E1 -9982.192,E2 -9982.192} C_VEL
LIN {X 0,Y 425.702,Z 405.904,A -85,B 0,C 180,E1 -9982.836,E2 -9982.836} C_VEL
LIN {X 0,Y 425.223,Z 401.588,A -85,B 0,C 180,E1 -9983.358,E2 -9983.358} C_VEL
LIN {X 0,Y 422.776,Z 394.133,A -85,B 0,C 180,E1 -9984.169,E2 -9984.169} C_VEL
LIN {X 0,Y 420.329,Z 386.104,A -85,B 0,C 180,E1 -9984.897,E2 -9984.897} C_VEL
LIN {X 0,Y 419.847,Z 380.759,A -85,B 0,C 180,E1 -9985.267,E2 -9985.267} C_VEL
LIN {X 0,Y 420.116,Z 370.976,A -85,B 0,C 180,E1 -9985.803,E2 -9985.803} C_VEL
LIN {X 0,Y 420.364,Z 358.711,A -85,B 0,C 180,E1 -9986.256,E2 -9986.256} C_VEL
LIN {X 0,Y 420.568,Z 338.288,A -85,B 0,C 180,E1 -9986.647,E2 -9986.647} C_VEL
LIN {X 0,Y 420.951,Z 294.256,A -85,B 0,C 180,E1 -9987.399,E2 -9987.399} C_VEL
LIN {X 0,Y 418.386,Z 279.839,A -85,B 0,C 180,E1 -9987.744,E2 -9987.744} C_VEL
LIN {X 0,Y 418.661,Z 270.943,A -85,B 0,C 180,E1 -9990,E2 -9990} C_VEL
LIN {X 0,Y 418.478,Z 268.173,A -85,B 0,C 180,E1 -9990.782,E2 -9990.782} C_VEL
LIN {X 0,Y 418.474,Z 268.17,A -85,B 0,C 180,E1 -9992.888,E2 -9992.888} C_VEL
LIN {X 0,Y 418.455,Z 268.171,A -85,B 0,C 180,E1 -9996.752,E2 -9996.752} C_VEL
LIN {X 0,Y 418.305,Z 268.19,A -85,B 0,C 180,E1 -9999.672,E2 -9999.672} C_VEL
LIN {X 0,Y 418.31,Z 268.19,A -85,B 0,C 180,E1 -10003.002,E2 -10003.002} C_VEL
LIN {X 0,Y 418.278,Z 268.192,A -85,B 0,C 180,E1 -10006.737,E2 -10006.737} C_VEL
LIN {X 0,Y 418.236,Z 268.199,A -85,B 0,C 180,E1 -10009.792,E2 -10009.792} C_VEL
LIN {X 0,Y 418.204,Z 268.201,A -85,B 0,C 180,E1 -10012.738,E2 -10012.738} C_VEL
LIN {X 0,Y 418.204,Z 268.202,A -85,B 0,C 180,E1 -10015.909,E2 -10015.909} C_VEL
LIN {X 0,Y 418.229,Z 268.2,A -85,B 0,C 180,E1 -10019.165,E2 -10019.165} C_VEL
LIN {X 0,Y 418.228,Z 268.198,A -85,B 0,C 180,E1 -10022.847,E2 -10022.847} C_VEL
LIN {X 0,Y 418.216,Z 268.199,A -85,B 0,C 180,E1 -10026.24,E2 -10026.24} C_VEL
LIN {X 0,Y 418.174,Z 268.21,A -85,B 0,C 180,E1 -10029.691,E2 -10029.691} C_VEL
LIN {X 0,Y 418.197,Z 268.202,A -85,B 0,C 180,E1 -10032.323,E2 -10032.323} C_VEL
LIN {X 0,Y 418.213,Z 268.2,A -85,B 0,C 180,E1 -10035.112,E2 -10035.112} C_VEL
LIN {X 0,Y 418.218,Z 268.205,A -85,B 0,C 180,E1 -10037.77,E2 -10037.77} C_VEL
LIN {X 0,Y 418.223,Z 268.198,A -85,B 0,C 180,E1 -10040.625,E2 -10040.625} C_VEL
LIN {X 0,Y 418.225,Z 268.202,A -85,B 0,C 180,E1 -10043.979,E2 -10043.979} C_VEL
LIN {X 0,Y 418.242,Z 268.197,A -85,B 0,C 180,E1 -10047.16,E2 -10047.16} C_VEL
LIN {X 0,Y 418.248,Z 268.195,A -85,B 0,C 180,E1 -10050.842,E2 -10050.842} C_VEL
LIN {X 0,Y 418.224,Z 268.202,A -85,B 0,C 180,E1 -10054.097,E2 -10054.097} C_VEL
LIN {X 0,Y 418.223,Z 268.199,A -85,B 0,C 180,E1 -10057.267,E2 -10057.267} C_VEL
LIN {X 0,Y 418.276,Z 268.194,A -85,B 0,C 180,E1 -10060.368,E2 -10060.368} C_VEL
LIN {X 0,Y 418.356,Z 268.315,A -85,B 0,C 180,E1 -10062.819,E2 -10062.819} C_VEL
LIN {X 0,Y 418.264,Z 278.685,A -85,B 0,C 180,E1 -10065.405,E2 -10065.405} C_VEL
LIN {X 0,Y 418.268,Z 279.535,A -85,B 0,C 180,E1 -10065.558,E2 -10065.558} C_VEL
LIN {X 0,Y 420.584,Z 295.353,A -85,B 0,C 180,E1 -10065.953,E2 -10065.953} C_VEL
LIN {X 0,Y 419.778,Z 357.101,A -85,B 0,C 180,E1 -10067.248,E2 -10067.248} C_VEL
LIN {X 0,Y 419.55,Z 367.315,A -85,B 0,C 180,E1 -10067.61,E2 -10067.61} C_VEL
LIN {X 0,Y 419.302,Z 376.992,A -85,B 0,C 180,E1 -10068.094,E2 -10068.094} C_VEL
LIN {X 0,Y 419.095,Z 387.112,A -85,B 0,C 180,E1 -10068.762,E2 -10068.762} C_VEL
LIN {X 0,Y 418.71,Z 396.824,A -85,B 0,C 180,E1 -10069.608,E2 -10069.608} C_VEL
LIN {X 0,Y 418.402,Z 404.647,A -85,B 0,C 180,E1 -10070.456,E2 -10070.456} C_VEL
LIN {X 0,Y 418.01,Z 412.849,A -85,B 0,C 180,E1 -10071.544,E2 -10071.544} C_VEL
LIN {X 0,Y 417.795,Z 420.392,A -85,B 0,C 180,E1 -10072.804,E2 -10072.804} C_VEL
LIN {X 0,Y 417.571,Z 424.841,A -85,B 0,C 180,E1 -10073.723,E2 -10073.723} C_VEL
LIN {X 0,Y 417.43,Z 428.725,A -85,B 0,C 180,E1 -10074.69,E2 -10074.69} C_VEL
LIN {X 0,Y 417.297,Z 433.173,A -85,B 0,C 180,E1 -10076.14,E2 -10076.14} C_VEL
LIN {X 0,Y 417.241,Z 435.427,A -85,B 0,C 180,E1 -10077.107,E2 -10077.107} C_VEL
LIN {X 0,Y 417.127,Z 437.1,A -85,B 0,C 180,E1 -10078.072,E2 -10078.072} C_VEL
LIN {X 0,Y 417.064,Z 438.163,A -85,B 0,C 180,E1 -10079.038,E2 -10079.038} C_VEL
LIN {X 0,Y 417.059,Z 438.677,A -85,B 0,C 180,E1 -10080.003,E2 -10080.003} C_VEL
LIN {X 0,Y 417.09,Z 438.678,A -85,B 0,C 180,E1 -10080.969,E2 -10080.969} C_VEL
LIN {X 0,Y 417.161,Z 438.166,A -85,B 0,C 180,E1 -10081.934,E2 -10081.934} C_VEL
LIN {X 0,Y 417.288,Z 437.132,A -85,B 0,C 180,E1 -10082.899,E2 -10082.899} C_VEL
LIN {X 0,Y 417.549,Z 434.433,A -85,B 0,C 180,E1 -10084.347,E2 -10084.347} C_VEL
LIN {X 0,Y 417.627,Z 431.961,A -85,B 0,C 180,E1 -10085.314,E2 -10085.314} C_VEL
LIN {X 0,Y 417.769,Z 428.85,A -85,B 0,C 180,E1 -10086.281,E2 -10086.281} C_VEL
LIN {X 0,Y 418.13,Z 424.31,A -85,B 0,C 180,E1 -10087.393,E2 -10087.393} C_VEL
LIN {X 0,Y 418.398,Z 418.99,A -85,B 0,C 180,E1 -10088.455,E2 -10088.455} C_VEL
LIN {X 0,Y 418.773,Z 413.1,A -85,B 0,C 180,E1 -10089.42,E2 -10089.42} C_VEL
LIN {X 0,Y 419.217,Z 405.952,A -85,B 0,C 180,E1 -10090.385,E2 -10090.385} C_VEL
LIN {X 0,Y 419.712,Z 397.182,A -85,B 0,C 180,E1 -10091.35,E2 -10091.35} C_VEL
LIN {X 0,Y 420.245,Z 387.352,A -85,B 0,C 180,E1 -10092.192,E2 -10092.192} C_VEL
LIN {X 0,Y 420.648,Z 377.255,A -85,B 0,C 180,E1 -10092.854,E2 -10092.854} C_VEL
LIN {X 0,Y 420.922,Z 367.597,A -85,B 0,C 180,E1 -10093.336,E2 -10093.336} C_VEL
LIN {X 0,Y 421.239,Z 355.655,A -85,B 0,C 180,E1 -10093.743,E2 -10093.743} C_VEL
LIN {X 0,Y 422.367,Z 295.008,A -85,B 0,C 180,E1 -10095.114,E2 -10095.114} C_VEL
LIN {X 0,Y 419.206,Z 281.294,A -85,B 0,C 180,E1 -10095.625,E2 -10095.625} C_VEL
LIN {X 0,Y 419.253,Z 273.328,A -85,B 0,C 180,E1 -10097.564,E2 -10097.564} C_VEL
LIN {X 0,Y 418.346,Z 268.195,A -85,B 0,C 180,E1 -10098.934,E2 -10098.934} C_VEL
LIN {X 0,Y 418.24,Z 268.202,A -85,B 0,C 180,E1 -10102.739,E2 -10102.739} C_VEL
LIN {X 0,Y 418.242,Z 268.203,A -85,B 0,C 180,E1 -10105.908,E2 -10105.908} C_VEL
LIN {X 0,Y 418.27,Z 268.195,A -85,B 0,C 180,E1 -10109.164,E2 -10109.164} C_VEL
LIN {X 0,Y 418.261,Z 268.198,A -85,B 0,C 180,E1 -10112.844,E2 -10112.844} C_VEL
LIN {X 0,Y 418.252,Z 268.201,A -85,B 0,C 180,E1 -10116.239,E2 -10116.239} C_VEL
LIN {X 0,Y 418.209,Z 268.202,A -85,B 0,C 180,E1 -10119.689,E2 -10119.689} C_VEL
LIN {X 0,Y 418.23,Z 268.201,A -85,B 0,C 180,E1 -10122.321,E2 -10122.321} C_VEL
LIN {X 0,Y 418.245,Z 268.197,A -85,B 0,C 180,E1 -10125.11,E2 -10125.11} C_VEL
LIN {X 0,Y 418.243,Z 268.195,A -85,B 0,C 180,E1 -10127.767,E2 -10127.767} C_VEL
LIN {X 0,Y 418.246,Z 268.196,A -85,B 0,C 180,E1 -10131.557,E2 -10131.557} C_VEL
LIN {X 0,Y 418.259,Z 268.196,A -85,B 0,C 180,E1 -10135.159,E2 -10135.159} C_VEL
LIN {X 0,Y 418.251,Z 268.197,A -85,B 0,C 180,E1 -10137.472,E2 -10137.472} C_VEL
LIN {X 0,Y 418.277,Z 268.194,A -85,B 0,C 180,E1 -10140.896,E2 -10140.896} C_VEL
LIN {X 0,Y 418.305,Z 268.192,A -85,B 0,C 180,E1 -10144.098,E2 -10144.098} C_VEL
LIN {X 0,Y 418.379,Z 268.393,A -85,B 0,C 180,E1 -10144.856,E2 -10144.856} C_VEL
LIN {X 0,Y 419.886,Z 277.893,A -85,B 0,C 180,E1 -10147.014,E2 -10147.014} C_VEL
LIN {X 0,Y 419.095,Z 293.624,A -85,B 0,C 180,E1 -10150.404,E2 -10150.404} C_VEL
LIN {X 0,Y 418.249,Z 313.205,A -85,B 0,C 180,E1 -10154.575,E2 -10154.575} C_VEL
LIN {X 0,Y 420.585,Z 330.84,A -85,B 0,C 180,E1 -10155.15,E2 -10155.15} C_VEL
LIN {X 0,Y 421.422,Z 341.211,A -85,B 0,C 180,E1 -10155.444,E2 -10155.444} C_VEL
LIN {X 0,Y 420.341,Z 396.456,A -85,B 0,C 180,E1 -10156.709,E2 -10156.709} C_VEL
LIN {X 0,Y 419.835,Z 408.478,A -85,B 0,C 180,E1 -10157.185,E2 -10157.185} C_VEL
LIN {X 0,Y 419.353,Z 419.43,A -85,B 0,C 180,E1 -10157.785,E2 -10157.785} C_VEL
LIN {X 0,Y 418.913,Z 429.334,A -85,B 0,C 180,E1 -10158.508,E2 -10158.508} C_VEL
LIN {X 0,Y 418.408,Z 439.466,A -85,B 0,C 180,E1 -10159.475,E2 -10159.475} C_VEL
LIN {X 0,Y 417.95,Z 448.276,A -85,B 0,C 180,E1 -10160.564,E2 -10160.564} C_VEL
LIN {X 0,Y 417.651,Z 454.64,A -85,B 0,C 180,E1 -10161.533,E2 -10161.533} C_VEL
LIN {X 0,Y 417.446,Z 461.112,A -85,B 0,C 180,E1 -10162.746,E2 -10162.746} C_VEL
LIN {X 0,Y 417.152,Z 467.18,A -85,B 0,C 180,E1 -10164.198,E2 -10164.198} C_VEL
LIN {X 0,Y 417.092,Z 471.571,A -85,B 0,C 180,E1 -10165.651,E2 -10165.651} C_VEL
LIN {X 0,Y 417.123,Z 474.643,A -85,B 0,C 180,E1 -10167.102,E2 -10167.102} C_VEL
LIN {X 0,Y 417.097,Z 476.038,A -85,B 0,C 180,E1 -10168.069,E2 -10168.069} C_VEL
LIN {X 0,Y 417.059,Z 476.941,A -85,B 0,C 180,E1 -10169.034,E2 -10169.034} C_VEL
LIN {X 0,Y 417.057,Z 477.261,A -85,B 0,C 180,E1 -10170,E2 -10170} C_VEL
LIN {X 0,Y 417.048,Z 477.06,A -85,B 0,C 180,E1 -10170.965,E2 -10170.965} C_VEL
LIN {X 0,Y 417.095,Z 476.399,A -85,B 0,C 180,E1 -10171.931,E2 -10171.931} C_VEL
LIN {X 0,Y 417.09,Z 475.262,A -85,B 0,C 180,E1 -10172.897,E2 -10172.897} C_VEL
LIN {X 0,Y 417.092,Z 472.47,A -85,B 0,C 180,E1 -10174.348,E2 -10174.348} C_VEL
LIN {X 0,Y 417.155,Z 468.424,A -85,B 0,C 180,E1 -10175.801,E2 -10175.801} C_VEL
LIN {X 0,Y 417.467,Z 462.984,A -85,B 0,C 180,E1 -10177.253,E2 -10177.253} C_VEL
LIN {X 0,Y 417.703,Z 457.057,A -85,B 0,C 180,E1 -10178.466,E2 -10178.466} C_VEL
LIN {X 0,Y 418.177,Z 449.554,A -85,B 0,C 180,E1 -10179.675,E2 -10179.675} C_VEL
LIN {X 0,Y 418.645,Z 442.168,A -85,B 0,C 180,E1 -10180.641,E2 -10180.641} C_VEL
LIN {X 0,Y 419.111,Z 434.27,A -85,B 0,C 180,E1 -10181.486,E2 -10181.486} C_VEL
LIN {X 0,Y 419.737,Z 424.438,A -85,B 0,C 180,E1 -10182.326,E2 -10182.326} C_VEL
LIN {X 0,Y 420.306,Z 413.002,A -85,B 0,C 180,E1 -10183.046,E2 -10183.046} C_VEL
LIN {X 0,Y 420.734,Z 402.969,A -85,B 0,C 180,E1 -10183.493,E2 -10183.493} C_VEL
LIN {X 0,Y 421.072,Z 393.905,A -85,B 0,C 180,E1 -10183.767,E2 -10183.767} C_VEL
LIN {X 0,Y 421.501,Z 339.326,A -85,B 0,C 180,E1 -10184.739,E2 -10184.739} C_VEL
LIN {X 0,Y 419.43,Z 322.852,A -85,B 0,C 180,E1 -10185.117,E2 -10185.117} C_VEL
LIN {X 0,Y 418.392,Z 315.888,A -85,B 0,C 180,E1 -10185.316,E2 -10185.316} C_VEL
LIN {X 0,Y 419.144,Z 299.491,A -85,B 0,C 180,E1 -10188.831,E2 -10188.831} C_VEL
LIN {X 0,Y 420.026,Z 284.351,A -85,B 0,C 180,E1 -10192.115,E2 -10192.115} C_VEL
LIN {X 0,Y 420.26,Z 278.944,A -85,B 0,C 180,E1 -10193.308,E2 -10193.308} C_VEL
LIN {X 0,Y 418.337,Z 268.189,A -85,B 0,C 180,E1 -10195.899,E2 -10195.899} C_VEL
LIN {X 0,Y 418.272,Z 268.197,A -85,B 0,C 180,E1 -10199.161,E2 -10199.161} C_VEL
LIN {X 0,Y 418.258,Z 268.193,A -85,B 0,C 180,E1 -10202.841,E2 -10202.841} C_VEL
LIN {X 0,Y 418.251,Z 268.192,A -85,B 0,C 180,E1 -10206.237,E2 -10206.237} C_VEL
LIN {X 0,Y 418.236,Z 268.202,A -85,B 0,C 180,E1 -10209.683,E2 -10209.683} C_VEL
LIN {X 0,Y 418.231,Z 268.198,A -85,B 0,C 180,E1 -10212.319,E2 -10212.319} C_VEL
LIN {X 0,Y 418.243,Z 268.197,A -85,B 0,C 180,E1 -10215.107,E2 -10215.107} C_VEL
LIN {X 0,Y 418.241,Z 268.199,A -85,B 0,C 180,E1 -10217.765,E2 -10217.765} C_VEL
LIN {X 0,Y 418.245,Z 268.197,A -85,B 0,C 180,E1 -10221.555,E2 -10221.555} C_VEL
LIN {X 0,Y 418.265,Z 268.191,A -85,B 0,C 180,E1 -10225.157,E2 -10225.157} C_VEL
LIN {X 0,Y 418.252,Z 268.2,A -85,B 0,C 180,E1 -10227.47,E2 -10227.47} C_VEL
LIN {X 0,Y 418.27,Z 268.192,A -85,B 0,C 180,E1 -10230.895,E2 -10230.895} C_VEL
LIN {X 0,Y 418.244,Z 268.197,A -85,B 0,C 180,E1 -10234.092,E2 -10234.092} C_VEL
LIN {X 0,Y 418.238,Z 268.198,A -85,B 0,C 180,E1 -10237.261,E2 -10237.261} C_VEL
LIN {X 0,Y 418.289,Z 268.191,A -85,B 0,C 180,E1 -10240.362,E2 -10240.362} C_VEL
LIN {X 0,Y 418.321,Z 268.184,A -85,B 0,C 180,E1 -10243.402,E2 -10243.402} C_VEL
LIN {X 0,Y 418.351,Z 268.18,A -85,B 0,C 180,E1 -10246.997,E2 -10246.997} C_VEL
LIN {X 0,Y 418.343,Z 268.183,A -85,B 0,C 180,E1 -10250.326,E2 -10250.326} C_VEL
LIN {X 0,Y 418.49,Z 268.161,A -85,B 0,C 180,E1 -10253.246,E2 -10253.246} C_VEL
LIN {X 0,Y 418.332,Z 268.177,A -85,B 0,C 180,E1 -10255.179,E2 -10255.179} C_VEL
LIN {X 0,Y 418.54,Z 268.16,A -85,B 0,C 180,E1 -10258.072,E2 -10258.072} C_VEL
LIN {X 0,Y 418.667,Z 268.139,A -85,B 0,C 180,E1 -10259.997,E2 -10259.997} C_VEL
LIN {X 0,Y 418.492,Z 268.163,A -85,B 0,C 180,E1 -10262.885,E2 -10262.885} C_VEL
LIN {X 0,Y 418.454,Z 268.167,A -85,B 0,C 180,E1 -10266.526,E2 -10266.526} C_VEL
LIN {X 0,Y 418.335,Z 268.184,A -85,B 0,C 180,E1 -10269.668,E2 -10269.668} C_VEL
LIN {X 0,Y 418.341,Z 268.184,A -85,B 0,C 180,E1 -10272.997,E2 -10272.997} C_VEL
LIN {X 0,Y 418.305,Z 268.19,A -85,B 0,C 180,E1 -10276.732,E2 -10276.732} C_VEL
LIN {X 0,Y 418.261,Z 268.193,A -85,B 0,C 180,E1 -10279.787,E2 -10279.787} C_VEL
LIN {X 0,Y 418.227,Z 268.201,A -85,B 0,C 180,E1 -10282.733,E2 -10282.733} C_VEL
LIN {X 0,Y 418.258,Z 268.194,A -85,B 0,C 180,E1 -10285.9,E2 -10285.9} C_VEL
LIN {X 0,Y 418.25,Z 268.196,A -85,B 0,C 180,E1 -10289.158,E2 -10289.158} C_VEL
LIN {X 0,Y 418.24,Z 268.201,A -85,B 0,C 180,E1 -10292.84,E2 -10292.84} C_VEL
LIN {X 0,Y 418.226,Z 268.192,A -85,B 0,C 180,E1 -10296.235,E2 -10296.235} C_VEL
LIN {X 0,Y 418.228,Z 268.196,A -85,B 0,C 180,E1 -10299.679,E2 -10299.679} C_VEL
LIN {X 0,Y 418.261,Z 268.198,A -85,B 0,C 180,E1 -10302.326,E2 -10302.326} C_VEL
LIN {X 0,Y 418.251,Z 268.2,A -85,B 0,C 180,E1 -10305.111,E2 -10305.111} C_VEL
LIN {X 0,Y 418.267,Z 268.194,A -85,B 0,C 180,E1 -10307.77,E2 -10307.77} C_VEL
LIN {X 0,Y 418.239,Z 268.201,A -85,B 0,C 180,E1 -10311.557,E2 -10311.557} C_VEL
LIN {X 0,Y 418.266,Z 268.266,A -85,B 0,C 180,E1 -10314.792,E2 -10314.792} C_VEL
LIN {X 0,Y 418.999,Z 273.418,A -85,B 0,C 180,E1 -10316.137,E2 -10316.137} C_VEL
LIN {X 0,Y 418.836,Z 280.004,A -85,B 0,C 180,E1 -10317.773,E2 -10317.773} C_VEL
LIN {X 0,Y 421.988,Z 295.206,A -85,B 0,C 180,E1 -10318.186,E2 -10318.186} C_VEL
LIN {X 0,Y 421.32,Z 356.882,A -85,B 0,C 180,E1 -10319.279,E2 -10319.279} C_VEL
LIN {X 0,Y 421.099,Z 367.184,A -85,B 0,C 180,E1 -10319.609,E2 -10319.609} C_VEL
LIN {X 0,Y 420.768,Z 378.85,A -85,B 0,C 180,E1 -10320.184,E2 -10320.184} C_VEL
LIN {X 0,Y 420.384,Z 387.839,A -85,B 0,C 180,E1 -10320.798,E2 -10320.798} C_VEL
LIN {X 0,Y 419.918,Z 396.123,A -85,B 0,C 180,E1 -10321.511,E2 -10321.511} C_VEL
LIN {X 0,Y 419.468,Z 402.924,A -85,B 0,C 180,E1 -10322.22,E2 -10322.22} C_VEL
LIN {X 0,Y 419.036,Z 409.715,A -85,B 0,C 180,E1 -10323.074,E2 -10323.074} C_VEL
LIN {X 0,Y 418.561,Z 416.505,A -85,B 0,C 180,E1 -10324.115,E2 -10324.115} C_VEL
LIN {X 0,Y 418.213,Z 422.067,A -85,B 0,C 180,E1 -10325.158,E2 -10325.158} C_VEL
LIN {X 0,Y 417.878,Z 426.617,A -85,B 0,C 180,E1 -10326.194,E2 -10326.194} C_VEL
LIN {X 0,Y 417.614,Z 430.321,A -85,B 0,C 180,E1 -10327.228,E2 -10327.228} C_VEL
LIN {X 0,Y 417.438,Z 433.289,A -85,B 0,C 180,E1 -10328.26,E2 -10328.26} C_VEL
LIN {X 0,Y 417.298,Z 435.597,A -85,B 0,C 180,E1 -10329.288,E2 -10329.288} C_VEL
LIN {X 0,Y 417.105,Z 437.638,A -85,B 0,C 180,E1 -10330.645,E2 -10330.645} C_VEL
LIN {X 0,Y 417.065,Z 438.304,A -85,B 0,C 180,E1 -10331.327,E2 -10331.327} C_VEL
LIN {X 0,Y 417.002,Z 438.794,A -85,B 0,C 180,E1 -10332.34,E2 -10332.34} C_VEL
LIN {X 0,Y 417.046,Z 438.598,A -85,B 0,C 180,E1 -10333.835,E2 -10333.835} C_VEL
LIN {X 0,Y 417.057,Z 437.173,A -85,B 0,C 180,E1 -10335.359,E2 -10335.359} C_VEL
LIN {X 0,Y 417.214,Z 434.419,A -85,B 0,C 180,E1 -10336.856,E2 -10336.856} C_VEL
LIN {X 0,Y 417.395,Z 431.549,A -85,B 0,C 180,E1 -10337.968,E2 -10337.968} C_VEL
LIN {X 0,Y 417.502,Z 428.786,A -85,B 0,C 180,E1 -10338.838,E2 -10338.838} C_VEL
LIN {X 0,Y 417.768,Z 423.794,A -85,B 0,C 180,E1 -10340.071,E2 -10340.071} C_VEL
LIN {X 0,Y 418.11,Z 417.475,A -85,B 0,C 180,E1 -10341.299,E2 -10341.299} C_VEL
LIN {X 0,Y 418.428,Z 411.292,A -85,B 0,C 180,E1 -10342.278,E2 -10342.278} C_VEL
LIN {X 0,Y 418.703,Z 405.668,A -85,B 0,C 180,E1 -10343.03,E2 -10343.03} C_VEL
LIN {X 0,Y 419.091,Z 398.173,A -85,B 0,C 180,E1 -10343.863,E2 -10343.863} C_VEL
LIN {X 0,Y 419.485,Z 390.128,A -85,B 0,C 180,E1 -10344.593,E2 -10344.593} C_VEL
LIN {X 0,Y 419.819,Z 381.816,A -85,B 0,C 180,E1 -10345.199,E2 -10345.199} C_VEL
LIN {X 0,Y 419.847,Z 380.759,A -85,B 0,C 180,E1 -10345.267,E2 -10345.267} C_VEL
LIN {X 0,Y 419.594,Z 376.292,A -85,B 0,C 180,E1 -10345.551,E2 -10345.551} C_VEL
LIN {X 0,Y 416.754,Z 366.512,A -85,B 0,C 180,E1 -10346.089,E2 -10346.089} C_VEL
LIN {X 0,Y 414.153,Z 357.357,A -85,B 0,C 180,E1 -10346.467,E2 -10346.467} C_VEL
LIN {X 0,Y 413.528,Z 351.586,A -85,B 0,C 180,E1 -10346.613,E2 -10346.613} C_VEL
LIN {X 0,Y 413.955,Z 294.842,A -85,B 0,C 180,E1 -10347.598,E2 -10347.598} C_VEL
LIN {X 0,Y 411.38,Z 280.147,A -85,B 0,C 180,E1 -10347.95,E2 -10347.95} C_VEL
LIN {X 0,Y 411.571,Z 270.302,A -85,B 0,C 180,E1 -10350.489,E2 -10350.489} C_VEL
LIN {X 0,Y 411.443,Z 269.049,A -85,B 0,C 180,E1 -10350.857,E2 -10350.857} C_VEL
LIN {X 0,Y 411.429,Z 269.048,A -85,B 0,C 180,E1 -10352.938,E2 -10352.938} C_VEL
LIN {X 0,Y 411.422,Z 269.048,A -85,B 0,C 180,E1 -10356.868,E2 -10356.868} C_VEL
LIN {X 0,Y 411.257,Z 269.067,A -85,B 0,C 180,E1 -10359.84,E2 -10359.84} C_VEL
LIN {X 0,Y 411.27,Z 269.069,A -85,B 0,C 180,E1 -10363.105,E2 -10363.105} C_VEL
LIN {X 0,Y 411.223,Z 269.072,A -85,B 0,C 180,E1 -10366.89,E2 -10366.89} C_VEL
LIN {X 0,Y 411.197,Z 269.074,A -85,B 0,C 180,E1 -10369.989,E2 -10369.989} C_VEL
LIN {X 0,Y 411.168,Z 269.08,A -85,B 0,C 180,E1 -10373.15,E2 -10373.15} C_VEL
LIN {X 0,Y 411.163,Z 269.077,A -85,B 0,C 180,E1 -10376.386,E2 -10376.386} C_VEL
LIN {X 0,Y 411.167,Z 269.081,A -85,B 0,C 180,E1 -10379.716,E2 -10379.716} C_VEL
LIN {X 0,Y 411.178,Z 269.078,A -85,B 0,C 180,E1 -10383.159,E2 -10383.159} C_VEL
LIN {X 0,Y 411.164,Z 269.077,A -85,B 0,C 180,E1 -10386.555,E2 -10386.555} C_VEL
LIN {X 0,Y 411.143,Z 269.086,A -85,B 0,C 180,E1 -10389.724,E2 -10389.724} C_VEL
LIN {X 0,Y 411.146,Z 269.081,A -85,B 0,C 180,E1 -10393.137,E2 -10393.137} C_VEL
LIN {X 0,Y 411.145,Z 269.084,A -85,B 0,C 180,E1 -10395.885,E2 -10395.885} C_VEL
LIN {X 0,Y 411.143,Z 269.08,A -85,B 0,C 180,E1 -10398.775,E2 -10398.775} C_VEL
LIN {X 0,Y 411.172,Z 269.08,A -85,B 0,C 180,E1 -10402.029,E2 -10402.029} C_VEL
LIN {X 0,Y 411.189,Z 269.08,A -85,B 0,C 180,E1 -10405.67,E2 -10405.67} C_VEL
LIN {X 0,Y 411.175,Z 269.077,A -85,B 0,C 180,E1 -10409.156,E2 -10409.156} C_VEL
LIN {X 0,Y 411.177,Z 269.077,A -85,B 0,C 180,E1 -10412.521,E2 -10412.521} C_VEL
LIN {X 0,Y 411.194,Z 269.079,A -85,B 0,C 180,E1 -10415.787,E2 -10415.787} C_VEL
LIN {X 0,Y 411.188,Z 269.075,A -85,B 0,C 180,E1 -10418.97,E2 -10418.97} C_VEL
LIN {X 0,Y 411.318,Z 269.12,A -85,B 0,C 180,E1 -10422.772,E2 -10422.772} C_VEL
LIN {X 0,Y 411.224,Z 278.608,A -85,B 0,C 180,E1 -10425.15,E2 -10425.15} C_VEL
LIN {X 0,Y 411.221,Z 279.483,A -85,B 0,C 180,E1 -10425.367,E2 -10425.367} C_VEL
LIN {X 0,Y 413.6,Z 295.583,A -85,B 0,C 180,E1 -10425.785,E2 -10425.785} C_VEL
LIN {X 0,Y 412.765,Z 357.582,A -85,B 0,C 180,E1 -10427.122,E2 -10427.122} C_VEL
LIN {X 0,Y 412.559,Z 367.014,A -85,B 0,C 180,E1 -10427.459,E2 -10427.459} C_VEL
LIN {X 0,Y 412.304,Z 376.82,A -85,B 0,C 180,E1 -10427.951,E2 -10427.951} C_VEL
LIN {X 0,Y 412.019,Z 387.862,A -85,B 0,C 180,E1 -10428.691,E2 -10428.691} C_VEL
LIN {X 0,Y 411.647,Z 397.466,A -85,B 0,C 180,E1 -10429.552,E2 -10429.552} C_VEL
LIN {X 0,Y 411.332,Z 405.248,A -85,B 0,C 180,E1 -10430.414,E2 -10430.414} C_VEL
LIN {X 0,Y 410.956,Z 412.57,A -85,B 0,C 180,E1 -10431.397,E2 -10431.397} C_VEL
LIN {X 0,Y 410.723,Z 420.283,A -85,B 0,C 180,E1 -10432.68,E2 -10432.68} C_VEL
LIN {X 0,Y 410.427,Z 426.792,A -85,B 0,C 180,E1 -10434.106,E2 -10434.106} C_VEL
LIN {X 0,Y 410.285,Z 430.388,A -85,B 0,C 180,E1 -10435.09,E2 -10435.09} C_VEL
LIN {X 0,Y 410.221,Z 434.509,A -85,B 0,C 180,E1 -10436.566,E2 -10436.566} C_VEL
LIN {X 0,Y 410.057,Z 437.319,A -85,B 0,C 180,E1 -10438.039,E2 -10438.039} C_VEL
LIN {X 0,Y 409.986,Z 438.414,A -85,B 0,C 180,E1 -10439.021,E2 -10439.021} C_VEL
LIN {X 0,Y 409.979,Z 438.983,A -85,B 0,C 180,E1 -10440.003,E2 -10440.003} C_VEL
LIN {X 0,Y 410.012,Z 439.04,A -85,B 0,C 180,E1 -10440.985,E2 -10440.985} C_VEL
LIN {X 0,Y 410.09,Z 438.583,A -85,B 0,C 180,E1 -10441.967,E2 -10441.967} C_VEL
LIN {X 0,Y 410.228,Z 437.6,A -85,B 0,C 180,E1 -10442.949,E2 -10442.949} C_VEL
LIN {X 0,Y 410.507,Z 434.962,A -85,B 0,C 180,E1 -10444.422,E2 -10444.422} C_VEL
LIN {X 0,Y 410.551,Z 431.057,A -85,B 0,C 180,E1 -10445.898,E2 -10445.898} C_VEL
LIN {X 0,Y 411.047,Z 426.426,A -85,B 0,C 180,E1 -10447.181,E2 -10447.181} C_VEL
LIN {X 0,Y 411.437,Z 419.722,A -85,B 0,C 180,E1 -10448.599,E2 -10448.599} C_VEL
LIN {X 0,Y 411.829,Z 413.888,A -85,B 0,C 180,E1 -10449.581,E2 -10449.581} C_VEL
LIN {X 0,Y 412.298,Z 406.822,A -85,B 0,C 180,E1 -10450.562,E2 -10450.562} C_VEL
LIN {X 0,Y 412.825,Z 398.205,A -85,B 0,C 180,E1 -10451.542,E2 -10451.542} C_VEL
LIN {X 0,Y 413.478,Z 387.045,A -85,B 0,C 180,E1 -10452.519,E2 -10452.519} C_VEL
LIN {X 0,Y 413.871,Z 377.919,A -85,B 0,C 180,E1 -10453.13,E2 -10453.13} C_VEL
LIN {X 0,Y 414.183,Z 368.407,A -85,B 0,C 180,E1 -10453.62,E2 -10453.62} C_VEL
LIN {X 0,Y 414.484,Z 357.511,A -85,B 0,C 180,E1 -10454.016,E2 -10454.016} C_VEL
LIN {X 0,Y 415.816,Z 296.434,A -85,B 0,C 180,E1 -10455.434,E2 -10455.434} C_VEL
LIN {X 0,Y 412.746,Z 283.268,A -85,B 0,C 180,E1 -10455.961,E2 -10455.961} C_VEL
LIN {X 0,Y 412.327,Z 281.483,A -85,B 0,C 180,E1 -10456.051,E2 -10456.051} C_VEL
LIN {X 0,Y 412.308,Z 274.132,A -85,B 0,C 180,E1 -10457.87,E2 -10457.87} C_VEL
LIN {X 0,Y 411.281,Z 269.073,A -85,B 0,C 180,E1 -10459.272,E2 -10459.272} C_VEL
LIN {X 0,Y 411.203,Z 269.076,A -85,B 0,C 180,E1 -10463.15,E2 -10463.15} C_VEL
LIN {X 0,Y 411.202,Z 269.078,A -85,B 0,C 180,E1 -10466.386,E2 -10466.386} C_VEL
LIN {X 0,Y 411.207,Z 269.076,A -85,B 0,C 180,E1 -10469.715,E2 -10469.715} C_VEL
LIN {X 0,Y 411.214,Z 269.074,A -85,B 0,C 180,E1 -10473.158,E2 -10473.158} C_VEL
LIN {X 0,Y 411.201,Z 269.078,A -85,B 0,C 180,E1 -10476.554,E2 -10476.554} C_VEL
LIN {X 0,Y 411.178,Z 269.078,A -85,B 0,C 180,E1 -10479.722,E2 -10479.722} C_VEL
LIN {X 0,Y 411.179,Z 269.077,A -85,B 0,C 180,E1 -10483.135,E2 -10483.135} C_VEL
LIN {X 0,Y 411.176,Z 269.077,A -85,B 0,C 180,E1 -10485.882,E2 -10485.882} C_VEL
LIN {X 0,Y 411.167,Z 269.081,A -85,B 0,C 180,E1 -10488.774,E2 -10488.774} C_VEL
LIN {X 0,Y 411.194,Z 269.076,A -85,B 0,C 180,E1 -10492.026,E2 -10492.026} C_VEL
LIN {X 0,Y 411.211,Z 269.074,A -85,B 0,C 180,E1 -10495.124,E2 -10495.124} C_VEL
LIN {X 0,Y 411.172,Z 269.079,A -85,B 0,C 180,E1 -10498.003,E2 -10498.003} C_VEL
LIN {X 0,Y 411.226,Z 269.074,A -85,B 0,C 180,E1 -10501.41,E2 -10501.41} C_VEL
LIN {X 0,Y 411.311,Z 269.224,A -85,B 0,C 180,E1 -10504.712,E2 -10504.712} C_VEL
LIN {X 0,Y 412.879,Z 278.905,A -85,B 0,C 180,E1 -10506.952,E2 -10506.952} C_VEL
LIN {X 0,Y 412.056,Z 294.27,A -85,B 0,C 180,E1 -10510.314,E2 -10510.314} C_VEL
LIN {X 0,Y 411.228,Z 312.001,A -85,B 0,C 180,E1 -10514.157,E2 -10514.157} C_VEL
LIN {X 0,Y 413.799,Z 330.414,A -85,B 0,C 180,E1 -10514.787,E2 -10514.787} C_VEL
LIN {X 0,Y 414.736,Z 342.132,A -85,B 0,C 180,E1 -10515.13,E2 -10515.13} C_VEL
LIN {X 0,Y 413.578,Z 395.612,A -85,B 0,C 180,E1 -10516.393,E2 -10516.393} C_VEL
LIN {X 0,Y 413.012,Z 408.344,A -85,B 0,C 180,E1 -10516.907,E2 -10516.907} C_VEL
LIN {X 0,Y 412.5,Z 417.761,A -85,B 0,C 180,E1 -10517.453,E2 -10517.453} C_VEL
LIN {X 0,Y 411.999,Z 427.553,A -85,B 0,C 180,E1 -10518.188,E2 -10518.188} C_VEL
LIN {X 0,Y 411.454,Z 437.651,A -85,B 0,C 180,E1 -10519.17,E2 -10519.17} C_VEL
LIN {X 0,Y 411.027,Z 445.903,A -85,B 0,C 180,E1 -10520.155,E2 -10520.155} C_VEL
LIN {X 0,Y 410.597,Z 454.121,A -85,B 0,C 180,E1 -10521.386,E2 -10521.386} C_VEL
LIN {X 0,Y 410.384,Z 460.625,A -85,B 0,C 180,E1 -10522.62,E2 -10522.62} C_VEL
LIN {X 0,Y 410.061,Z 466.71,A -85,B 0,C 180,E1 -10524.097,E2 -10524.097} C_VEL
LIN {X 0,Y 410.022,Z 471.152,A -85,B 0,C 180,E1 -10525.576,E2 -10525.576} C_VEL
LIN {X 0,Y 410.021,Z 474.25,A -85,B 0,C 180,E1 -10527.052,E2 -10527.052} C_VEL
LIN {X 0,Y 410.026,Z 475.673,A -85,B 0,C 180,E1 -10528.035,E2 -10528.035} C_VEL
LIN {X 0,Y 409.982,Z 476.593,A -85,B 0,C 180,E1 -10529.018,E2 -10529.018} C_VEL
LIN {X 0,Y 409.976,Z 476.921,A -85,B 0,C 180,E1 -10530,E2 -10530} C_VEL
LIN {X 0,Y 409.971,Z 476.746,A -85,B 0,C 180,E1 -10530.982,E2 -10530.982} C_VEL
LIN {X 0,Y 410.023,Z 476.11,A -85,B 0,C 180,E1 -10531.964,E2 -10531.964} C_VEL
LIN {X 0,Y 409.987,Z 474.997,A -85,B 0,C 180,E1 -10532.948,E2 -10532.948} C_VEL
LIN {X 0,Y 410.022,Z 472.232,A -85,B 0,C 180,E1 -10534.424,E2 -10534.424} C_VEL
LIN {X 0,Y 410.079,Z 468.213,A -85,B 0,C 180,E1 -10535.902,E2 -10535.902} C_VEL
LIN {X 0,Y 410.274,Z 464.738,A -85,B 0,C 180,E1 -10536.887,E2 -10536.887} C_VEL
LIN {X 0,Y 410.539,Z 459.368,A -85,B 0,C 180,E1 -10538.119,E2 -10538.119} C_VEL
LIN {X 0,Y 410.855,Z 454.103,A -85,B 0,C 180,E1 -10539.104,E2 -10539.104} C_VEL
LIN {X 0,Y 411.307,Z 447.782,A -85,B 0,C 180,E1 -10540.087,E2 -10540.087} C_VEL
LIN {X 0,Y 411.914,Z 439.089,A -85,B 0,C 180,E1 -10541.191,E2 -10541.191} C_VEL
LIN {X 0,Y 412.568,Z 429.091,A -85,B 0,C 180,E1 -10542.169,E2 -10542.169} C_VEL
LIN {X 0,Y 412.971,Z 421.251,A -85,B 0,C 180,E1 -10542.781,E2 -10542.781} C_VEL
LIN {X 0,Y 413.484,Z 412.281,A -85,B 0,C 180,E1 -10543.328,E2 -10543.328} C_VEL
LIN {X 0,Y 413.921,Z 402.367,A -85,B 0,C 180,E1 -10543.773,E2 -10543.773} C_VEL
LIN {X 0,Y 414.252,Z 393.318,A -85,B 0,C 180,E1 -10544.048,E2 -10544.048} C_VEL
LIN {X 0,Y 414.749,Z 340.319,A -85,B 0,C 180,E1 -10545.007,E2 -10545.007} C_VEL
LIN {X 0,Y 412.593,Z 323.275,A -85,B 0,C 180,E1 -10545.409,E2 -10545.409} C_VEL
LIN {X 0,Y 411.396,Z 315.523,A -85,B 0,C 180,E1 -10545.635,E2 -10545.635} C_VEL
LIN {X 0,Y 412.223,Z 299.371,A -85,B 0,C 180,E1 -10549.159,E2 -10549.159} C_VEL
LIN {X 0,Y 413.247,Z 283.096,A -85,B 0,C 180,E1 -10552.762,E2 -10552.762} C_VEL
LIN {X 0,Y 413.155,Z 279.252,A -85,B 0,C 180,E1 -10553.642,E2 -10553.642} C_VEL
LIN {X 0,Y 411.291,Z 269.066,A -85,B 0,C 180,E1 -10556.172,E2 -10556.172} C_VEL
LIN {X 0,Y 411.208,Z 269.073,A -85,B 0,C 180,E1 -10559.712,E2 -10559.712} C_VEL
LIN {X 0,Y 411.212,Z 269.073,A -85,B 0,C 180,E1 -10563.155,E2 -10563.155} C_VEL
LIN {X 0,Y 411.199,Z 269.07,A -85,B 0,C 180,E1 -10566.551,E2 -10566.551} C_VEL
LIN {X 0,Y 411.202,Z 269.078,A -85,B 0,C 180,E1 -10569.724,E2 -10569.724} C_VEL
LIN {X 0,Y 411.178,Z 269.08,A -85,B 0,C 180,E1 -10573.133,E2 -10573.133} C_VEL
LIN {X 0,Y 411.174,Z 269.08,A -85,B 0,C 180,E1 -10575.88,E2 -10575.88} C_VEL
LIN {X 0,Y 411.165,Z 269.078,A -85,B 0,C 180,E1 -10578.771,E2 -10578.771} C_VEL
LIN {X 0,Y 411.194,Z 269.076,A -85,B 0,C 180,E1 -10582.024,E2 -10582.024} C_VEL
LIN {X 0,Y 411.212,Z 269.073,A -85,B 0,C 180,E1 -10585.665,E2 -10585.665} C_VEL
LIN {X 0,Y 411.195,Z 269.071,A -85,B 0,C 180,E1 -10589.151,E2 -10589.151} C_VEL
LIN {X 0,Y 411.195,Z 269.072,A -85,B 0,C 180,E1 -10592.515,E2 -10592.515} C_VEL
LIN {X 0,Y 411.219,Z 269.077,A -85,B 0,C 180,E1 -10595.782,E2 -10595.782} C_VEL
LIN {X 0,Y 411.202,Z 269.066,A -85,B 0,C 180,E1 -10598.964,E2 -10598.964} C_VEL
LIN {X 0,Y 411.251,Z 269.067,A -85,B 0,C 180,E1 -10602.082,E2 -10602.082} C_VEL
LIN {X 0,Y 411.264,Z 269.061,A -85,B 0,C 180,E1 -10605.145,E2 -10605.145} C_VEL
LIN {X 0,Y 411.287,Z 269.058,A -85,B 0,C 180,E1 -10608.165,E2 -10608.165} C_VEL
LIN {X 0,Y 411.443,Z 269.043,A -85,B 0,C 180,E1 -10612.186,E2 -10612.186} C_VEL
LIN {X 0,Y 411.474,Z 269.034,A -85,B 0,C 180,E1 -10614.115,E2 -10614.115} C_VEL
LIN {X 0,Y 411.509,Z 269.036,A -85,B 0,C 180,E1 -10618.039,E2 -10618.039} C_VEL
LIN {X 0,Y 411.636,Z 269.015,A -85,B 0,C 180,E1 -10619.997,E2 -10619.997} C_VEL
LIN {X 0,Y 411.449,Z 269.04,A -85,B 0,C 180,E1 -10622.934,E2 -10622.934} C_VEL
LIN {X 0,Y 411.42,Z 269.045,A -85,B 0,C 180,E1 -10626.864,E2 -10626.864} C_VEL
LIN {X 0,Y 411.287,Z 269.063,A -85,B 0,C 180,E1 -10629.835,E2 -10629.835} C_VEL
LIN {X 0,Y 411.3,Z 269.061,A -85,B 0,C 180,E1 -10633.101,E2 -10633.101} C_VEL
LIN {X 0,Y 411.25,Z 269.068,A -85,B 0,C 180,E1 -10636.885,E2 -10636.885} C_VEL
LIN {X 0,Y 411.221,Z 269.072,A -85,B 0,C 180,E1 -10639.983,E2 -10639.983} C_VEL
LIN {X 0,Y 411.192,Z 269.074,A -85,B 0,C 180,E1 -10643.144,E2 -10643.144} C_VEL
LIN {X 0,Y 411.225,Z 269.076,A -85,B 0,C 180,E1 -10646.377,E2 -10646.377} C_VEL
LIN {X 0,Y 411.185,Z 269.075,A -85,B 0,C 180,E1 -10649.709,E2 -10649.709} C_VEL
LIN {X 0,Y 411.189,Z 269.076,A -85,B 0,C 180,E1 -10653.152,E2 -10653.152} C_VEL
LIN {X 0,Y 411.174,Z 269.073,A -85,B 0,C 180,E1 -10656.549,E2 -10656.549} C_VEL
LIN {X 0,Y 411.192,Z 269.073,A -85,B 0,C 180,E1 -10659.724,E2 -10659.724} C_VEL
LIN {X 0,Y 411.199,Z 269.075,A -85,B 0,C 180,E1 -10663.124,E2 -10663.124} C_VEL
LIN {X 0,Y 411.216,Z 269.074,A -85,B 0,C 180,E1 -10665.867,E2 -10665.867} C_VEL
LIN {X 0,Y 411.187,Z 269.078,A -85,B 0,C 180,E1 -10669.497,E2 -10669.497} C_VEL
LIN {X 0,Y 411.178,Z 269.081,A -85,B 0,C 180,E1 -10672.025,E2 -10672.025} C_VEL
LIN {X 0,Y 411.213,Z 269.101,A -85,B 0,C 180,E1 -10674.556,E2 -10674.556} C_VEL
LIN {X 0,Y 412.044,Z 274.59,A -85,B 0,C 180,E1 -10676.015,E2 -10676.015} C_VEL
LIN {X 0,Y 411.891,Z 280.332,A -85,B 0,C 180,E1 -10677.462,E2 -10677.462} C_VEL
LIN {X 0,Y 415.246,Z 296.298,A -85,B 0,C 180,E1 -10677.905,E2 -10677.905} C_VEL
LIN {X 0,Y 414.522,Z 357.236,A -85,B 0,C 180,E1 -10679.003,E2 -10679.003} C_VEL
LIN {X 0,Y 414.311,Z 367.55,A -85,B 0,C 180,E1 -10679.339,E2 -10679.339} C_VEL
LIN {X 0,Y 413.984,Z 378.422,A -85,B 0,C 180,E1 -10679.874,E2 -10679.874} C_VEL
LIN {X 0,Y 413.49,Z 388.913,A -85,B 0,C 180,E1 -10680.608,E2 -10680.608} C_VEL
LIN {X 0,Y 413.049,Z 396.44,A -85,B 0,C 180,E1 -10681.271,E2 -10681.271} C_VEL
LIN {X 0,Y 412.495,Z 404.544,A -85,B 0,C 180,E1 -10682.15,E2 -10682.15} C_VEL
LIN {X 0,Y 412.119,Z 410.025,A -85,B 0,C 180,E1 -10682.859,E2 -10682.859} C_VEL
LIN {X 0,Y 411.605,Z 416.811,A -85,B 0,C 180,E1 -10683.917,E2 -10683.917} C_VEL
LIN {X 0,Y 411.189,Z 422.6,A -85,B 0,C 180,E1 -10685.025,E2 -10685.025} C_VEL
LIN {X 0,Y 410.801,Z 427.936,A -85,B 0,C 180,E1 -10686.294,E2 -10686.294} C_VEL
LIN {X 0,Y 410.421,Z 432.983,A -85,B 0,C 180,E1 -10687.869,E2 -10687.869} C_VEL
LIN {X 0,Y 410.258,Z 435.412,A -85,B 0,C 180,E1 -10688.916,E2 -10688.916} C_VEL
LIN {X 0,Y 410.031,Z 437.903,A -85,B 0,C 180,E1 -10690.496,E2 -10690.496} C_VEL
LIN {X 0,Y 409.919,Z 439.041,A -85,B 0,C 180,E1 -10692.025,E2 -10692.025} C_VEL
LIN {X 0,Y 409.947,Z 438.953,A -85,B 0,C 180,E1 -10693.731,E2 -10693.731} C_VEL
LIN {X 0,Y 409.967,Z 437.806,A -85,B 0,C 180,E1 -10695.1,E2 -10695.1} C_VEL
LIN {X 0,Y 410.112,Z 435.348,A -85,B 0,C 180,E1 -10696.624,E2 -10696.624} C_VEL
LIN {X 0,Y 410.328,Z 431.487,A -85,B 0,C 180,E1 -10698.139,E2 -10698.139} C_VEL
LIN {X 0,Y 410.583,Z 426.228,A -85,B 0,C 180,E1 -10699.646,E2 -10699.646} C_VEL
LIN {X 0,Y 410.882,Z 420.571,A -85,B 0,C 180,E1 -10700.897,E2 -10700.897} C_VEL
LIN {X 0,Y 411.343,Z 412.633,A -85,B 0,C 180,E1 -10702.251,E2 -10702.251} C_VEL
LIN {X 0,Y 411.725,Z 405.168,A -85,B 0,C 180,E1 -10703.261,E2 -10703.261} C_VEL
LIN {X 0,Y 412.088,Z 398.543,A -85,B 0,C 180,E1 -10704.004,E2 -10704.004} C_VEL
LIN {X 0,Y 412.511,Z 390.502,A -85,B 0,C 180,E1 -10704.746,E2 -10704.746} C_VEL
LIN {X 0,Y 412.856,Z 382.203,A -85,B 0,C 180,E1 -10705.362,E2 -10705.362} C_VEL
LIN {X 0,Y 413.057,Z 373.836,A -85,B 0,C 180,E1 -10705.853,E2 -10705.853} C_VEL
LIN {X 0,Y 413.318,Z 364.683,A -85,B 0,C 180,E1 -10706.253,E2 -10706.253} C_VEL
LIN {X 0,Y 413.513,Z 355.291,A -85,B 0,C 180,E1 -10706.529,E2 -10706.529} C_VEL
LIN {X 0,Y 413.528,Z 351.586,A -85,B 0,C 180,E1 -10706.613,E2 -10706.613} C_VEL
LIN {X 0,Y 412.92,Z 345.78,A -85,B 0,C 180,E1 -10706.741,E2 -10706.741} C_VEL
LIN {X 0,Y 407.487,Z 327.019,A -85,B 0,C 180,E1 -10707.223,E2 -10707.223} C_VEL
LIN {X 0,Y 406.925,Z 321.203,A -85,B 0,C 180,E1 -10707.342,E2 -10707.342} C_VEL
LIN {X 0,Y 406.963,Z 295.393,A -85,B 0,C 180,E1 -10707.804,E2 -10707.804} C_VEL
LIN {X 0,Y 404.389,Z 280.451,A -85,B 0,C 180,E1 -10708.164,E2 -10708.164} C_VEL
LIN {X 0,Y 404.579,Z 271.515,A -85,B 0,C 180,E1 -10710.498,E2 -10710.498} C_VEL
LIN {X 0,Y 404.405,Z 269.926,A -85,B 0,C 180,E1 -10710.934,E2 -10710.934} C_VEL
LIN {X 0,Y 404.387,Z 269.926,A -85,B 0,C 180,E1 -10712.989,E2 -10712.989} C_VEL
LIN {X 0,Y 404.369,Z 269.928,A -85,B 0,C 180,E1 -10716.988,E2 -10716.988} C_VEL
LIN {X 0,Y 404.223,Z 269.942,A -85,B 0,C 180,E1 -10720.013,E2 -10720.013} C_VEL
LIN {X 0,Y 404.232,Z 269.947,A -85,B 0,C 180,E1 -10723.213,E2 -10723.213} C_VEL
LIN {X 0,Y 404.182,Z 269.95,A -85,B 0,C 180,E1 -10727.009,E2 -10727.009} C_VEL
LIN {X 0,Y 404.13,Z 269.953,A -85,B 0,C 180,E1 -10730.354,E2 -10730.354} C_VEL
LIN {X 0,Y 404.129,Z 269.959,A -85,B 0,C 180,E1 -10733.577,E2 -10733.577} C_VEL
LIN {X 0,Y 404.102,Z 269.958,A -85,B 0,C 180,E1 -10736.884,E2 -10736.884} C_VEL
LIN {X 0,Y 404.114,Z 269.955,A -85,B 0,C 180,E1 -10740.288,E2 -10740.288} C_VEL
LIN {X 0,Y 404.116,Z 269.959,A -85,B 0,C 180,E1 -10743.815,E2 -10743.815} C_VEL
LIN {X 0,Y 404.107,Z 269.957,A -85,B 0,C 180,E1 -10746.877,E2 -10746.877} C_VEL
LIN {X 0,Y 404.091,Z 269.96,A -85,B 0,C 180,E1 -10750.078,E2 -10750.078} C_VEL
LIN {X 0,Y 404.126,Z 269.955,A -85,B 0,C 180,E1 -10753.087,E2 -10753.087} C_VEL
LIN {X 0,Y 404.126,Z 269.958,A -85,B 0,C 180,E1 -10755.929,E2 -10755.929} C_VEL
LIN {X 0,Y 404.098,Z 269.958,A -85,B 0,C 180,E1 -10758.638,E2 -10758.638} C_VEL
LIN {X 0,Y 404.13,Z 269.957,A -85,B 0,C 180,E1 -10761.497,E2 -10761.497} C_VEL
LIN {X 0,Y 404.167,Z 269.949,A -85,B 0,C 180,E1 -10764.988,E2 -10764.988} C_VEL
LIN {X 0,Y 404.125,Z 269.956,A -85,B 0,C 180,E1 -10768.446,E2 -10768.446} C_VEL
LIN {X 0,Y 404.144,Z 269.952,A -85,B 0,C 180,E1 -10770.867,E2 -10770.867} C_VEL
LIN {X 0,Y 404.139,Z 269.956,A -85,B 0,C 180,E1 -10774.235,E2 -10774.235} C_VEL
LIN {X 0,Y 404.159,Z 269.952,A -85,B 0,C 180,E1 -10777.512,E2 -10777.512} C_VEL
LIN {X 0,Y 404.159,Z 269.951,A -85,B 0,C 180,E1 -10780.711,E2 -10780.711} C_VEL
LIN {X 0,Y 404.293,Z 270.049,A -85,B 0,C 180,E1 -10782.75,E2 -10782.75} C_VEL
LIN {X 0,Y 404.194,Z 279.606,A -85,B 0,C 180,E1 -10785.159,E2 -10785.159} C_VEL
LIN {X 0,Y 406.633,Z 296.578,A -85,B 0,C 180,E1 -10785.629,E2 -10785.629} C_VEL
LIN {X 0,Y 405.753,Z 357.923,A -85,B 0,C 180,E1 -10786.991,E2 -10786.991} C_VEL
LIN {X 0,Y 405.513,Z 367.987,A -85,B 0,C 180,E1 -10787.365,E2 -10787.365} C_VEL
LIN {X 0,Y 405.255,Z 377.611,A -85,B 0,C 180,E1 -10787.865,E2 -10787.865} C_VEL
LIN {X 0,Y 404.95,Z 388.496,A -85,B 0,C 180,E1 -10788.618,E2 -10788.618} C_VEL
LIN {X 0,Y 404.583,Z 398.023,A -85,B 0,C 180,E1 -10789.494,E2 -10789.494} C_VEL
LIN {X 0,Y 404.26,Z 405.764,A -85,B 0,C 180,E1 -10790.371,E2 -10790.371} C_VEL
LIN {X 0,Y 403.845,Z 413.902,A -85,B 0,C 180,E1 -10791.497,E2 -10791.497} C_VEL
LIN {X 0,Y 403.631,Z 421.096,A -85,B 0,C 180,E1 -10792.751,E2 -10792.751} C_VEL
LIN {X 0,Y 403.342,Z 426.726,A -85,B 0,C 180,E1 -10794.002,E2 -10794.002} C_VEL
LIN {X 0,Y 403.17,Z 431.966,A -85,B 0,C 180,E1 -10795.504,E2 -10795.504} C_VEL
LIN {X 0,Y 403.073,Z 435.768,A -85,B 0,C 180,E1 -10797.005,E2 -10797.005} C_VEL
LIN {X 0,Y 402.989,Z 437.5,A -85,B 0,C 180,E1 -10798.004,E2 -10798.004} C_VEL
LIN {X 0,Y 402.912,Z 438.654,A -85,B 0,C 180,E1 -10799.004,E2 -10799.004} C_VEL
LIN {X 0,Y 402.901,Z 439.287,A -85,B 0,C 180,E1 -10800.003,E2 -10800.003} C_VEL
LIN {X 0,Y 402.936,Z 439.406,A -85,B 0,C 180,E1 -10801.003,E2 -10801.003} C_VEL
LIN {X 0,Y 403.021,Z 439.007,A -85,B 0,C 180,E1 -10802.002,E2 -10802.002} C_VEL
LIN {X 0,Y 403.171,Z 438.057,A -85,B 0,C 180,E1 -10803.001,E2 -10803.001} C_VEL
LIN {X 0,Y 403.467,Z 435.491,A -85,B 0,C 180,E1 -10804.499,E2 -10804.499} C_VEL
LIN {X 0,Y 403.551,Z 433.121,A -85,B 0,C 180,E1 -10805.5,E2 -10805.5} C_VEL
LIN {X 0,Y 403.728,Z 430.09,A -85,B 0,C 180,E1 -10806.5,E2 -10806.5} C_VEL
LIN {X 0,Y 404.13,Z 426.001,A -85,B 0,C 180,E1 -10807.58,E2 -10807.58} C_VEL
LIN {X 0,Y 404.481,Z 420.523,A -85,B 0,C 180,E1 -10808.748,E2 -10808.748} C_VEL
LIN {X 0,Y 404.916,Z 414.802,A -85,B 0,C 180,E1 -10809.746,E2 -10809.746} C_VEL
LIN {X 0,Y 405.404,Z 407.865,A -85,B 0,C 180,E1 -10810.743,E2 -10810.743} C_VEL
LIN {X 0,Y 405.913,Z 400.514,A -85,B 0,C 180,E1 -10811.614,E2 -10811.614} C_VEL
LIN {X 0,Y 406.476,Z 391.501,A -85,B 0,C 180,E1 -10812.484,E2 -10812.484} C_VEL
LIN {X 0,Y 407.051,Z 380.711,A -85,B 0,C 180,E1 -10813.291,E2 -10813.291} C_VEL
LIN {X 0,Y 407.41,Z 370.564,A -85,B 0,C 180,E1 -10813.851,E2 -10813.851} C_VEL
LIN {X 0,Y 407.687,Z 361.306,A -85,B 0,C 180,E1 -10814.223,E2 -10814.223} C_VEL
LIN {X 0,Y 408.161,Z 345.948,A -85,B 0,C 180,E1 -10814.62,E2 -10814.62} C_VEL
LIN {X 0,Y 409.195,Z 297.148,A -85,B 0,C 180,E1 -10815.811,E2 -10815.811} C_VEL
LIN {X 0,Y 406.09,Z 284.087,A -85,B 0,C 180,E1 -10816.356,E2 -10816.356} C_VEL
LIN {X 0,Y 405.514,Z 281.776,A -85,B 0,C 180,E1 -10816.49,E2 -10816.49} C_VEL
LIN {X 0,Y 405.529,Z 276.613,A -85,B 0,C 180,E1 -10817.786,E2 -10817.786} C_VEL
LIN {X 0,Y 404.238,Z 269.95,A -85,B 0,C 180,E1 -10819.572,E2 -10819.572} C_VEL
LIN {X 0,Y 404.165,Z 269.953,A -85,B 0,C 180,E1 -10823.577,E2 -10823.577} C_VEL
LIN {X 0,Y 404.143,Z 269.958,A -85,B 0,C 180,E1 -10826.883,E2 -10826.883} C_VEL
LIN {X 0,Y 404.154,Z 269.957,A -85,B 0,C 180,E1 -10830.287,E2 -10830.287} C_VEL
LIN {X 0,Y 404.147,Z 269.955,A -85,B 0,C 180,E1 -10833.814,E2 -10833.814} C_VEL
LIN {X 0,Y 404.143,Z 269.957,A -85,B 0,C 180,E1 -10836.876,E2 -10836.876} C_VEL
LIN {X 0,Y 404.126,Z 269.959,A -85,B 0,C 180,E1 -10840.076,E2 -10840.076} C_VEL
LIN {X 0,Y 404.158,Z 269.952,A -85,B 0,C 180,E1 -10843.084,E2 -10843.084} C_VEL
LIN {X 0,Y 404.157,Z 269.952,A -85,B 0,C 180,E1 -10845.927,E2 -10845.927} C_VEL
LIN {X 0,Y 404.122,Z 269.959,A -85,B 0,C 180,E1 -10848.635,E2 -10848.635} C_VEL
LIN {X 0,Y 404.153,Z 269.952,A -85,B 0,C 180,E1 -10851.495,E2 -10851.495} C_VEL
LIN {X 0,Y 404.186,Z 269.951,A -85,B 0,C 180,E1 -10854.984,E2 -10854.984} C_VEL
LIN {X 0,Y 404.147,Z 269.953,A -85,B 0,C 180,E1 -10858.443,E2 -10858.443} C_VEL
LIN {X 0,Y 404.204,Z 269.948,A -85,B 0,C 180,E1 -10862.001,E2 -10862.001} C_VEL
LIN {X 0,Y 404.266,Z 270.009,A -85,B 0,C 180,E1 -10864.553,E2 -10864.553} C_VEL
LIN {X 0,Y 405.741,Z 278.857,A -85,B 0,C 180,E1 -10866.643,E2 -10866.643} C_VEL
LIN {X 0,Y 405.577,Z 285.443,A -85,B 0,C 180,E1 -10868.126,E2 -10868.126} C_VEL
LIN {X 0,Y 404.704,Z 300.775,A -85,B 0,C 180,E1 -10871.523,E2 -10871.523} C_VEL
LIN {X 0,Y 404.21,Z 310.68,A -85,B 0,C 180,E1 -10873.702,E2 -10873.702} C_VEL
LIN {X 0,Y 407.111,Z 330.114,A -85,B 0,C 180,E1 -10874.4,E2 -10874.4} C_VEL
LIN {X 0,Y 408.085,Z 342.817,A -85,B 0,C 180,E1 -10874.792,E2 -10874.792} C_VEL
LIN {X 0,Y 406.856,Z 395.111,A -85,B 0,C 180,E1 -10876.069,E2 -10876.069} C_VEL
LIN {X 0,Y 406.268,Z 407.309,A -85,B 0,C 180,E1 -10876.558,E2 -10876.558} C_VEL
LIN {X 0,Y 405.722,Z 416.855,A -85,B 0,C 180,E1 -10877.113,E2 -10877.113} C_VEL
LIN {X 0,Y 405.266,Z 425.19,A -85,B 0,C 180,E1 -10877.735,E2 -10877.735} C_VEL
LIN {X 0,Y 404.78,Z 433.311,A -85,B 0,C 180,E1 -10878.482,E2 -10878.482} C_VEL
LIN {X 0,Y 404.28,Z 442.134,A -85,B 0,C 180,E1 -10879.483,E2 -10879.483} C_VEL
LIN {X 0,Y 403.731,Z 450.78,A -85,B 0,C 180,E1 -10880.734,E2 -10880.734} C_VEL
LIN {X 0,Y 403.349,Z 457.688,A -85,B 0,C 180,E1 -10881.987,E2 -10881.987} C_VEL
LIN {X 0,Y 403.081,Z 463.78,A -85,B 0,C 180,E1 -10883.354,E2 -10883.354} C_VEL
LIN {X 0,Y 402.966,Z 467.842,A -85,B 0,C 180,E1 -10884.495,E2 -10884.495} C_VEL
LIN {X 0,Y 402.898,Z 471.892,A -85,B 0,C 180,E1 -10885.999,E2 -10885.999} C_VEL
LIN {X 0,Y 402.921,Z 473.857,A -85,B 0,C 180,E1 -10887,E2 -10887} C_VEL
LIN {X 0,Y 402.956,Z 475.308,A -85,B 0,C 180,E1 -10888.001,E2 -10888.001} C_VEL
LIN {X 0,Y 402.907,Z 476.242,A -85,B 0,C 180,E1 -10889,E2 -10889} C_VEL
LIN {X 0,Y 402.899,Z 476.581,A -85,B 0,C 180,E1 -10890,E2 -10890} C_VEL
LIN {X 0,Y 402.897,Z 476.431,A -85,B 0,C 180,E1 -10890.999,E2 -10890.999} C_VEL
LIN {X 0,Y 402.952,Z 475.82,A -85,B 0,C 180,E1 -10891.999,E2 -10891.999} C_VEL
LIN {X 0,Y 402.885,Z 474.732,A -85,B 0,C 180,E1 -10893,E2 -10893} C_VEL
LIN {X 0,Y 402.952,Z 471.994,A -85,B 0,C 180,E1 -10894.501,E2 -10894.501} C_VEL
LIN {X 0,Y 402.994,Z 468.007,A -85,B 0,C 180,E1 -10896.006,E2 -10896.006} C_VEL
LIN {X 0,Y 403.213,Z 464.569,A -85,B 0,C 180,E1 -10897.008,E2 -10897.008} C_VEL
LIN {X 0,Y 403.477,Z 459.241,A -85,B 0,C 180,E1 -10898.262,E2 -10898.262} C_VEL
LIN {X 0,Y 403.844,Z 454.025,A -85,B 0,C 180,E1 -10899.263,E2 -10899.263} C_VEL
LIN {X 0,Y 404.308,Z 447.762,A -85,B 0,C 180,E1 -10900.263,E2 -10900.263} C_VEL
LIN {X 0,Y 404.862,Z 440.161,A -85,B 0,C 180,E1 -10901.261,E2 -10901.261} C_VEL
LIN {X 0,Y 405.551,Z 430.744,A -85,B 0,C 180,E1 -10902.256,E2 -10902.256} C_VEL
LIN {X 0,Y 406.084,Z 421.619,A -85,B 0,C 180,E1 -10903.002,E2 -10903.002} C_VEL
LIN {X 0,Y 406.659,Z 411.649,A -85,B 0,C 180,E1 -10903.619,E2 -10903.619} C_VEL
LIN {X 0,Y 407.082,Z 402.076,A -85,B 0,C 180,E1 -10904.056,E2 -10904.056} C_VEL
LIN {X 0,Y 407.455,Z 393.672,A -85,B 0,C 180,E1 -10904.318,E2 -10904.318} C_VEL
LIN {X 0,Y 407.937,Z 353.098,A -85,B 0,C 180,E1 -10905.072,E2 -10905.072} C_VEL
LIN {X 0,Y 408.012,Z 341.198,A -85,B 0,C 180,E1 -10905.287,E2 -10905.287} C_VEL
LIN {X 0,Y 405.685,Z 322.826,A -85,B 0,C 180,E1 -10905.73,E2 -10905.73} C_VEL
LIN {X 0,Y 404.421,Z 315.329,A -85,B 0,C 180,E1 -10905.93,E2 -10905.93} C_VEL
LIN {X 0,Y 405.284,Z 299.276,A -85,B 0,C 180,E1 -10909.5,E2 -10909.5} C_VEL
LIN {X 0,Y 406.302,Z 284.171,A -85,B 0,C 180,E1 -10912.904,E2 -10912.904} C_VEL
LIN {X 0,Y 406.329,Z 281.391,A -85,B 0,C 180,E1 -10913.548,E2 -10913.548} C_VEL
LIN {X 0,Y 404.245,Z 269.944,A -85,B 0,C 180,E1 -10916.386,E2 -10916.386} C_VEL
LIN {X 0,Y 404.166,Z 269.951,A -85,B 0,C 180,E1 -10919.603,E2 -10919.603} C_VEL
LIN {X 0,Y 404.147,Z 269.949,A -85,B 0,C 180,E1 -10922.621,E2 -10922.621} C_VEL
LIN {X 0,Y 404.153,Z 269.951,A -85,B 0,C 180,E1 -10925.182,E2 -10925.182} C_VEL
LIN {X 0,Y 404.15,Z 269.954,A -85,B 0,C 180,E1 -10928.757,E2 -10928.757} C_VEL
LIN {X 0,Y 404.125,Z 269.958,A -85,B 0,C 180,E1 -10931.598,E2 -10931.598} C_VEL
LIN {X 0,Y 404.152,Z 269.949,A -85,B 0,C 180,E1 -10934.521,E2 -10934.521} C_VEL
LIN {X 0,Y 404.14,Z 269.955,A -85,B 0,C 180,E1 -10937.294,E2 -10937.294} C_VEL
LIN {X 0,Y 404.14,Z 269.953,A -85,B 0,C 180,E1 -10939.949,E2 -10939.949} C_VEL
LIN {X 0,Y 404.142,Z 269.954,A -85,B 0,C 180,E1 -10943.124,E2 -10943.124} C_VEL
LIN {X 0,Y 404.152,Z 269.953,A -85,B 0,C 180,E1 -10946.186,E2 -10946.186} C_VEL
LIN {X 0,Y 404.151,Z 269.952,A -85,B 0,C 180,E1 -10949.713,E2 -10949.713} C_VEL
LIN {X 0,Y 404.141,Z 269.951,A -85,B 0,C 180,E1 -10953.117,E2 -10953.117} C_VEL
LIN {X 0,Y 404.167,Z 269.95,A -85,B 0,C 180,E1 -10956.423,E2 -10956.423} C_VEL
LIN {X 0,Y 404.197,Z 269.947,A -85,B 0,C 180,E1 -10959.872,E2 -10959.872} C_VEL
LIN {X 0,Y 404.221,Z 269.938,A -85,B 0,C 180,E1 -10962.991,E2 -10962.991} C_VEL
LIN {X 0,Y 404.287,Z 269.932,A -85,B 0,C 180,E1 -10966.936,E2 -10966.936} C_VEL
LIN {X 0,Y 404.26,Z 269.935,A -85,B 0,C 180,E1 -10969.985,E2 -10969.985} C_VEL
LIN {X 0,Y 404.402,Z 269.915,A -85,B 0,C 180,E1 -10973.01,E2 -10973.01} C_VEL
LIN {X 0,Y 404.277,Z 269.927,A -85,B 0,C 180,E1 -10975.011,E2 -10975.011} C_VEL
LIN {X 0,Y 404.477,Z 269.913,A -85,B 0,C 180,E1 -10978.005,E2 -10978.005} C_VEL
LIN {X 0,Y 404.605,Z 269.89,A -85,B 0,C 180,E1 -10979.997,E2 -10979.997} C_VEL
LIN {X 0,Y 404.408,Z 269.917,A -85,B 0,C 180,E1 -10982.985,E2 -10982.985} C_VEL
LIN {X 0,Y 404.365,Z 269.923,A -85,B 0,C 180,E1 -10986.985,E2 -10986.985} C_VEL
LIN {X 0,Y 404.252,Z 269.939,A -85,B 0,C 180,E1 -10990.008,E2 -10990.008} C_VEL
LIN {X 0,Y 404.261,Z 269.938,A -85,B 0,C 180,E1 -10993.208,E2 -10993.208} C_VEL
LIN {X 0,Y 404.208,Z 269.944,A -85,B 0,C 180,E1 -10997.003,E2 -10997.003} C_VEL
LIN {X 0,Y 404.154,Z 269.951,A -85,B 0,C 180,E1 -11000.348,E2 -11000.348} C_VEL
LIN {X 0,Y 404.158,Z 269.95,A -85,B 0,C 180,E1 -11003.571,E2 -11003.571} C_VEL
LIN {X 0,Y 404.171,Z 269.948,A -85,B 0,C 180,E1 -11005.763,E2 -11005.763} C_VEL
LIN {X 0,Y 404.181,Z 269.949,A -85,B 0,C 180,E1 -11007.996,E2 -11007.996} C_VEL
LIN {X 0,Y 404.123,Z 269.953,A -85,B 0,C 180,E1 -11011.554,E2 -11011.554} C_VEL
LIN {X 0,Y 404.167,Z 269.943,A -85,B 0,C 180,E1 -11015.013,E2 -11015.013} C_VEL
LIN {X 0,Y 404.134,Z 269.958,A -85,B 0,C 180,E1 -11018.753,E2 -11018.753} C_VEL
LIN {X 0,Y 404.166,Z 269.951,A -85,B 0,C 180,E1 -11021.607,E2 -11021.607} C_VEL
